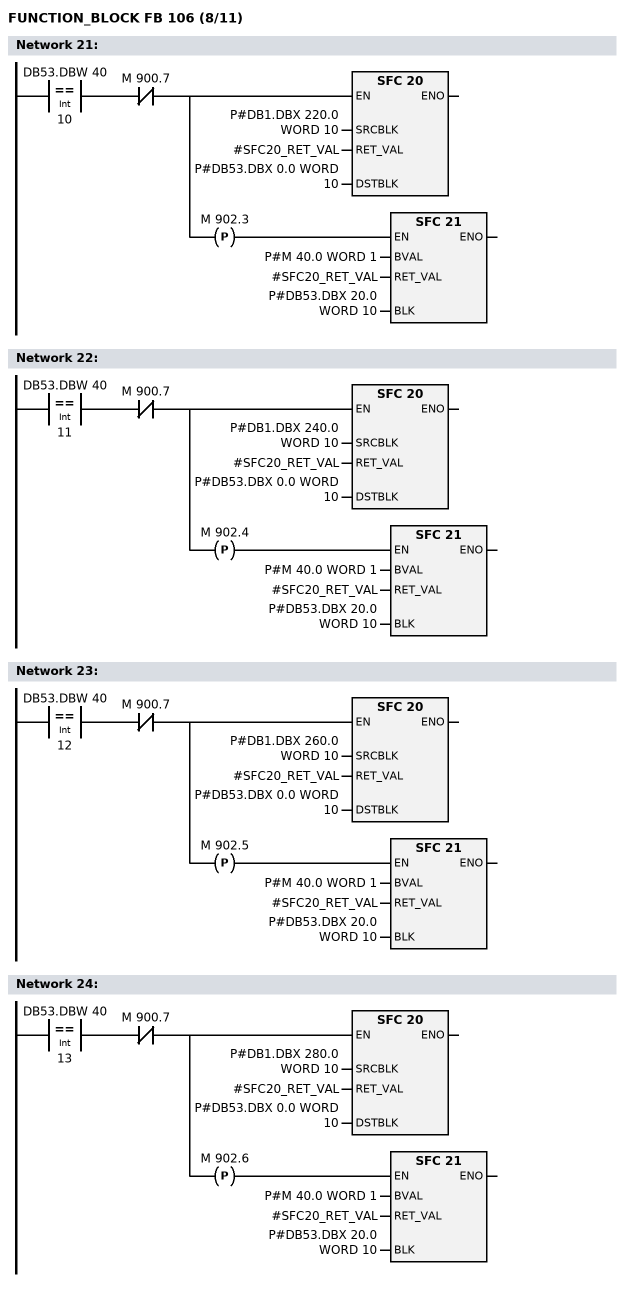

      A(    ;
      L     DB53.DBW   40;
      L     10;
      ==I   ;
      )     ;
      AN    M    900.7;
      =     L      0.0;
      A     L      0.0;
      JNB   _02d;
      CALL SFC   20 (
           SRCBLK                   := P#DB1.DBX 220.0 WORD 10,
           RET_VAL                  := #SFC20_RET_VAL,
           DSTBLK                   := P#DB53.DBX 0.0 WORD 10);
_02d: NOP   0;
      A     L      0.0;
      FP    M    902.3;
      JNB   _02e;
      CALL SFC   21 (
           BVAL                     := P#M 40.0 WORD 1,
           RET_VAL                  := #SFC20_RET_VAL,
           BLK                      := P#DB53.DBX 20.0 WORD 10);
_02e: NOP   0;
NETWORK
TITLE =

      A(    ;
      L     DB53.DBW   40;
      L     11;
      ==I   ;
      )     ;
      AN    M    900.7;
      =     L      0.0;
      A     L      0.0;
      JNB   _02f;
      CALL SFC   20 (
           SRCBLK                   := P#DB1.DBX 240.0 WORD 10,
           RET_VAL                  := #SFC20_RET_VAL,
           DSTBLK                   := P#DB53.DBX 0.0 WORD 10);
_02f: NOP   0;
      A     L      0.0;
      FP    M    902.4;
      JNB   _030;
      CALL SFC   21 (
           BVAL                     := P#M 40.0 WORD 1,
           RET_VAL                  := #SFC20_RET_VAL,
           BLK                      := P#DB53.DBX 20.0 WORD 10);
_030: NOP   0;
NETWORK
TITLE =

      A(    ;
      L     DB53.DBW   40;
      L     12;
      ==I   ;
      )     ;
      AN    M    900.7;
      =     L      0.0;
      A     L      0.0;
      JNB   _031;
      CALL SFC   20 (
           SRCBLK                   := P#DB1.DBX 260.0 WORD 10,
           RET_VAL                  := #SFC20_RET_VAL,
           DSTBLK                   := P#DB53.DBX 0.0 WORD 10);
_031: NOP   0;
      A     L      0.0;
      FP    M    902.5;
      JNB   _032;
      CALL SFC   21 (
           BVAL                     := P#M 40.0 WORD 1,
           RET_VAL                  := #SFC20_RET_VAL,
           BLK                      := P#DB53.DBX 20.0 WORD 10);
_032: NOP   0;
NETWORK
TITLE =

      A(    ;
      L     DB53.DBW   40;
      L     13;
      ==I   ;
      )     ;
      AN    M    900.7;
      =     L      0.0;
      A     L      0.0;
      JNB   _033;
      CALL SFC   20 (
           SRCBLK                   := P#DB1.DBX 280.0 WORD 10,
           RET_VAL                  := #SFC20_RET_VAL,
           DSTBLK                   := P#DB53.DBX 0.0 WORD 10);
_033: NOP   0;
      A     L      0.0;
      FP    M    902.6;
      JNB   _034;
      CALL SFC   21 (
           BVAL                     := P#M 40.0 WORD 1,
           RET_VAL                  := #SFC20_RET_VAL,
           BLK                      := P#DB53.DBX 20.0 WORD 10);
_034: NOP   0;
NETWORK
TITLE =
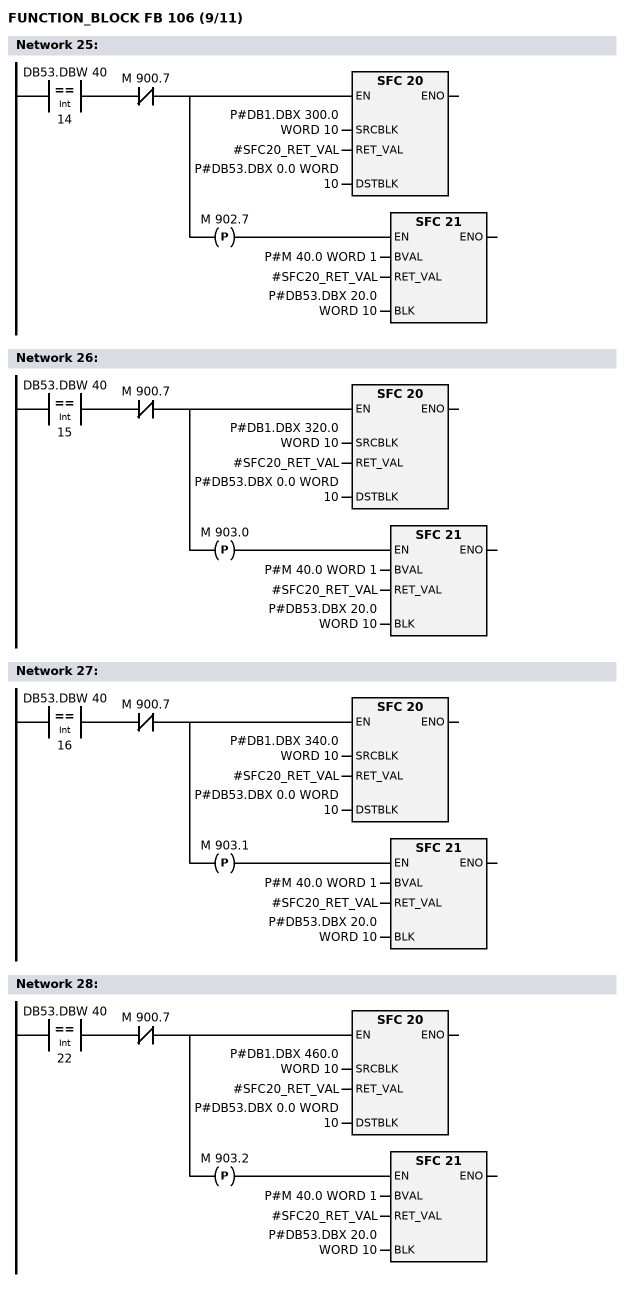

      A(    ;
      L     DB53.DBW   40;
      L     14;
      ==I   ;
      )     ;
      AN    M    900.7;
      =     L      0.0;
      A     L      0.0;
      JNB   _035;
      CALL SFC   20 (
           SRCBLK                   := P#DB1.DBX 300.0 WORD 10,
           RET_VAL                  := #SFC20_RET_VAL,
           DSTBLK                   := P#DB53.DBX 0.0 WORD 10);
_035: NOP   0;
      A     L      0.0;
      FP    M    902.7;
      JNB   _036;
      CALL SFC   21 (
           BVAL                     := P#M 40.0 WORD 1,
           RET_VAL                  := #SFC20_RET_VAL,
           BLK                      := P#DB53.DBX 20.0 WORD 10);
_036: NOP   0;
NETWORK
TITLE =

      A(    ;
      L     DB53.DBW   40;
      L     15;
      ==I   ;
      )     ;
      AN    M    900.7;
      =     L      0.0;
      A     L      0.0;
      JNB   _037;
      CALL SFC   20 (
           SRCBLK                   := P#DB1.DBX 320.0 WORD 10,
           RET_VAL                  := #SFC20_RET_VAL,
           DSTBLK                   := P#DB53.DBX 0.0 WORD 10);
_037: NOP   0;
      A     L      0.0;
      FP    M    903.0;
      JNB   _038;
      CALL SFC   21 (
           BVAL                     := P#M 40.0 WORD 1,
           RET_VAL                  := #SFC20_RET_VAL,
           BLK                      := P#DB53.DBX 20.0 WORD 10);
_038: NOP   0;
NETWORK
TITLE =

      A(    ;
      L     DB53.DBW   40;
      L     16;
      ==I   ;
      )     ;
      AN    M    900.7;
      =     L      0.0;
      A     L      0.0;
      JNB   _039;
      CALL SFC   20 (
           SRCBLK                   := P#DB1.DBX 340.0 WORD 10,
           RET_VAL                  := #SFC20_RET_VAL,
           DSTBLK                   := P#DB53.DBX 0.0 WORD 10);
_039: NOP   0;
      A     L      0.0;
      FP    M    903.1;
      JNB   _03a;
      CALL SFC   21 (
           BVAL                     := P#M 40.0 WORD 1,
           RET_VAL                  := #SFC20_RET_VAL,
           BLK                      := P#DB53.DBX 20.0 WORD 10);
_03a: NOP   0;
NETWORK
TITLE =

      A(    ;
      L     DB53.DBW   40;
      L     22;
      ==I   ;
      )     ;
      AN    M    900.7;
      =     L      0.0;
      A     L      0.0;
      JNB   _03b;
      CALL SFC   20 (
           SRCBLK                   := P#DB1.DBX 460.0 WORD 10,
           RET_VAL                  := #SFC20_RET_VAL,
           DSTBLK                   := P#DB53.DBX 0.0 WORD 10);
_03b: NOP   0;
      A     L      0.0;
      FP    M    903.2;
      JNB   _03c;
      CALL SFC   21 (
           BVAL                     := P#M 40.0 WORD 1,
           RET_VAL                  := #SFC20_RET_VAL,
           BLK                      := P#DB53.DBX 20.0 WORD 10);
_03c: NOP   0;
NETWORK
TITLE =
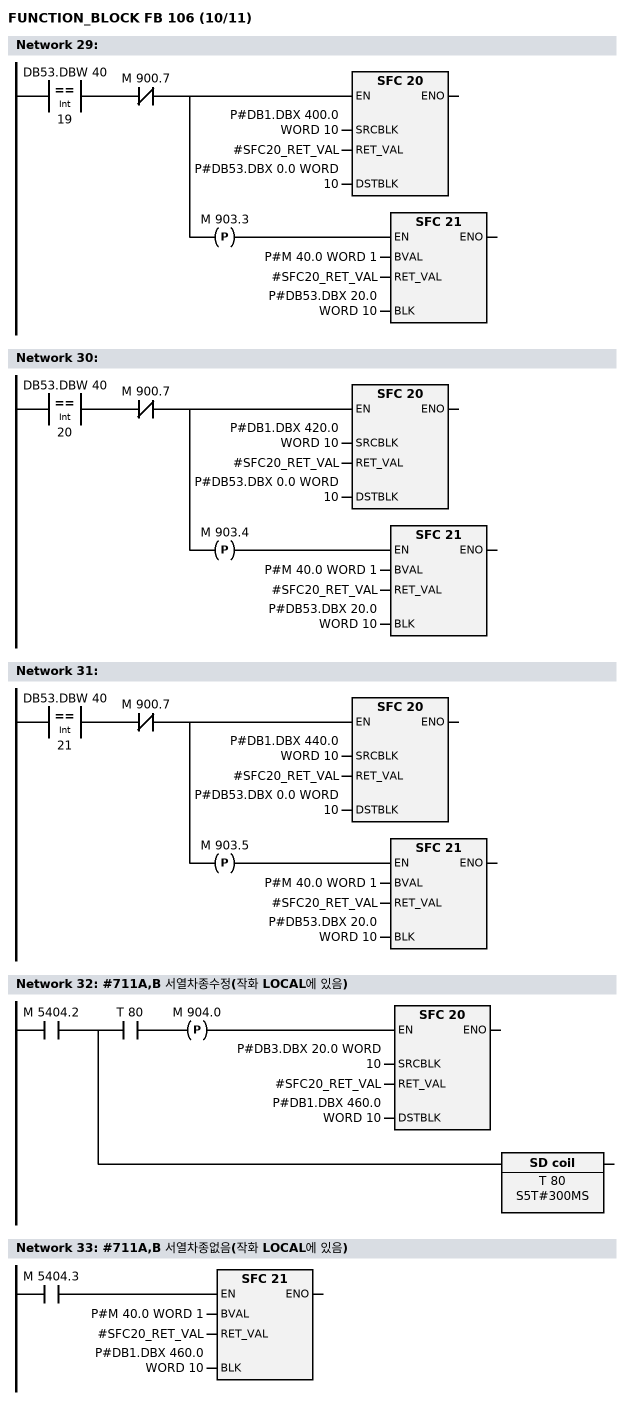

      A(    ;
      L     DB53.DBW   40;
      L     19;
      ==I   ;
      )     ;
      AN    M    900.7;
      =     L      0.0;
      A     L      0.0;
      JNB   _03d;
      CALL SFC   20 (
           SRCBLK                   := P#DB1.DBX 400.0 WORD 10,
           RET_VAL                  := #SFC20_RET_VAL,
           DSTBLK                   := P#DB53.DBX 0.0 WORD 10);
_03d: NOP   0;
      A     L      0.0;
      FP    M    903.3;
      JNB   _03e;
      CALL SFC   21 (
           BVAL                     := P#M 40.0 WORD 1,
           RET_VAL                  := #SFC20_RET_VAL,
           BLK                      := P#DB53.DBX 20.0 WORD 10);
_03e: NOP   0;
NETWORK
TITLE =

      A(    ;
      L     DB53.DBW   40;
      L     20;
      ==I   ;
      )     ;
      AN    M    900.7;
      =     L      0.0;
      A     L      0.0;
      JNB   _03f;
      CALL SFC   20 (
           SRCBLK                   := P#DB1.DBX 420.0 WORD 10,
           RET_VAL                  := #SFC20_RET_VAL,
           DSTBLK                   := P#DB53.DBX 0.0 WORD 10);
_03f: NOP   0;
      A     L      0.0;
      FP    M    903.4;
      JNB   _040;
      CALL SFC   21 (
           BVAL                     := P#M 40.0 WORD 1,
           RET_VAL                  := #SFC20_RET_VAL,
           BLK                      := P#DB53.DBX 20.0 WORD 10);
_040: NOP   0;
NETWORK
TITLE =

      A(    ;
      L     DB53.DBW   40;
      L     21;
      ==I   ;
      )     ;
      AN    M    900.7;
      =     L      0.0;
      A     L      0.0;
      JNB   _041;
      CALL SFC   20 (
           SRCBLK                   := P#DB1.DBX 440.0 WORD 10,
           RET_VAL                  := #SFC20_RET_VAL,
           DSTBLK                   := P#DB53.DBX 0.0 WORD 10);
_041: NOP   0;
      A     L      0.0;
      FP    M    903.5;
      JNB   _042;
      CALL SFC   21 (
           BVAL                     := P#M 40.0 WORD 1,
           RET_VAL                  := #SFC20_RET_VAL,
           BLK                      := P#DB53.DBX 20.0 WORD 10);
_042: NOP   0;
NETWORK
TITLE =#711A,B 서열차종수정(작화 LOCAL에 있음)

      A     M   5404.2;
      =     L      0.0;
      A     L      0.0;
      A     T     80;
      FP    M    904.0;
      JNB   _043;
      CALL SFC   20 (
           SRCBLK                   := P#DB3.DBX 20.0 WORD 10,
           RET_VAL                  := #SFC20_RET_VAL,
           DSTBLK                   := P#DB1.DBX 460.0 WORD 10);
_043: NOP   0;
      A     L      0.0;
      BLD   102;
      L     S5T#300MS;
      SD    T     80;
NETWORK
TITLE =#711A,B 서열차종없음(작화 LOCAL에 있음)

      A     M   5404.3;
      JNB   _044;
      CALL SFC   21 (
           BVAL                     := P#M 40.0 WORD 1,
           RET_VAL                  := #SFC20_RET_VAL,
           BLK                      := P#DB1.DBX 460.0 WORD 10);
_044: NOP   0;
NETWORK
TITLE =#711R1,R2 로보트 차종수정(작화 LOCAL에 있음)
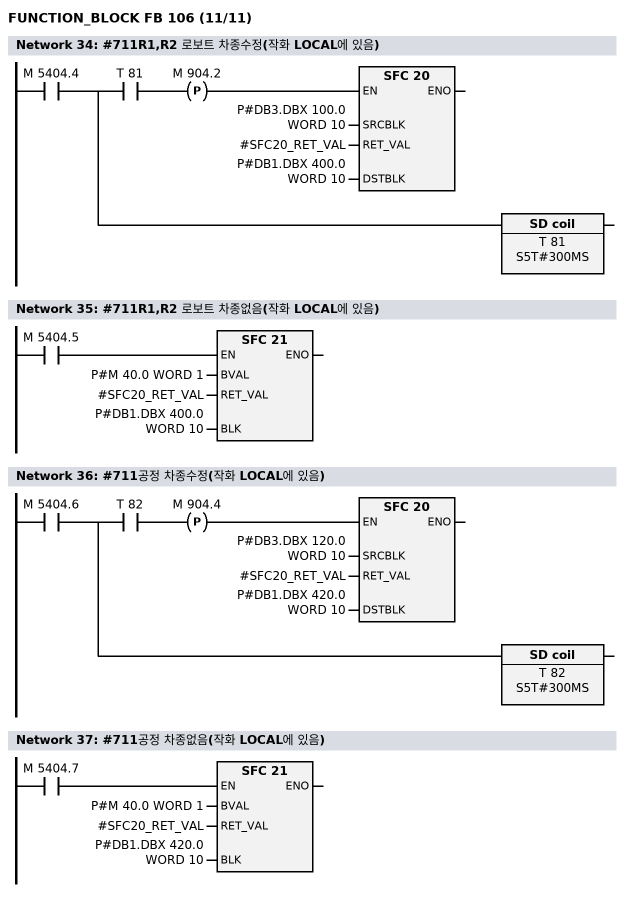

      A     M   5404.4;
      =     L      0.0;
      A     L      0.0;
      A     T     81;
      FP    M    904.2;
      JNB   _045;
      CALL SFC   20 (
           SRCBLK                   := P#DB3.DBX 100.0 WORD 10,
           RET_VAL                  := #SFC20_RET_VAL,
           DSTBLK                   := P#DB1.DBX 400.0 WORD 10);
_045: NOP   0;
      A     L      0.0;
      BLD   102;
      L     S5T#300MS;
      SD    T     81;
NETWORK
TITLE =#711R1,R2 로보트 차종없음(작화 LOCAL에 있음)

      A     M   5404.5;
      JNB   _046;
      CALL SFC   21 (
           BVAL                     := P#M 40.0 WORD 1,
           RET_VAL                  := #SFC20_RET_VAL,
           BLK                      := P#DB1.DBX 400.0 WORD 10);
_046: NOP   0;
NETWORK
TITLE =#711공정 차종수정(작화 LOCAL에 있음)

      A     M   5404.6;
      =     L      0.0;
      A     L      0.0;
      A     T     82;
      FP    M    904.4;
      JNB   _047;
      CALL SFC   20 (
           SRCBLK                   := P#DB3.DBX 120.0 WORD 10,
           RET_VAL                  := #SFC20_RET_VAL,
           DSTBLK                   := P#DB1.DBX 420.0 WORD 10);
_047: NOP   0;
      A     L      0.0;
      BLD   102;
      L     S5T#300MS;
      SD    T     82;
NETWORK
TITLE =#711공정 차종없음(작화 LOCAL에 있음)

      A     M   5404.7;
      JNB   _048;
      CALL SFC   21 (
           BVAL                     := P#M 40.0 WORD 1,
           RET_VAL                  := #SFC20_RET_VAL,
           BLK                      := P#DB1.DBX 420.0 WORD 10);
_048: NOP   0;
END_FUNCTION_BLOCK

DATA_BLOCK DB 106
TITLE =
VERSION : 0.0

 FB 106
BEGIN
   CAR_TYPE_MODIFY.Station := 0;
   CAR_TYPE_MODIFY.HMI_Disp_DB := 0;
   CAR_TYPE_MODIFY.HMI_Disp_Add := 0;
   CAR_TYPE_MODIFY.CType_DB := 0;
   CAR_TYPE_MODIFY.CType_Start_Add := 0;
   CAR_TYPE_MODIFY.Byte_per_Stn := 0;
   CAR_TYPE_MODIFY.M_Modify_OK := FALSE;
   CAR_TYPE_MODIFY.SS_CCR_On := FALSE;
   CAR_TYPE_MODIFY.PB_Set := FALSE;
   CAR_TYPE_MODIFY.PB_Reset := FALSE;
   CAR_TYPE_MODIFY.LP_CCR_On := FALSE;
   CAR_TYPE_MODIFY.LP_Modify_On := FALSE;
   CAR_TYPE_MODIFY.Source_Data := W#16#0;
   CAR_TYPE_MODIFY.Modify_Data := W#16#0;
   CAR_TYPE_MODIFY.Pre_Station := 0;
   CAR_TYPE_MODIFY.Station_PLS := FALSE;
   CAR_TYPE_MODIFY.Source_Add := 0;
   CAR_TYPE_MODIFY.SFC20_Ret := 0;
   CAR_TYPE_MODIFY.Fill_Source := W#16#0;
   SFC20_RET_VAL := 0;
   HMI_CAR_TYPE_V2.Stn_Vin_No := L#0;
   HMI_CAR_TYPE_V2.Stn_Bt_1Word := W#16#0;
   HMI_CAR_TYPE_V2.Stn_Bt_2Word := W#16#0;
   HMI_CAR_TYPE_V2.Stn_Bt_3Word := W#16#0;
   HMI_CAR_TYPE_V2.Stn_Bt_4Word := W#16#0;
   HMI_CAR_TYPE_V2.Stn_Bt_5Word_Sp := W#16#0;
   HMI_CAR_TYPE_V2.Stn_Bt_6Word_Sp := W#16#0;
   HMI_CAR_TYPE_V2.M_BType_On := FALSE;
   HMI_CAR_TYPE_V2.M_BType_None := FALSE;
   HMI_CAR_TYPE_V2.M_Bypass_BType := FALSE;
   HMI_CAR_TYPE_V2.M_BType_TL := FALSE;
   HMI_CAR_TYPE_V2.M_BType_LM := FALSE;
   HMI_CAR_TYPE_V2.M_BType_SP1 := FALSE;
   HMI_CAR_TYPE_V2.M_BType_SP2 := FALSE;
   HMI_CAR_TYPE_V2.M_BType_SP3 := FALSE;
   HMI_CAR_TYPE_V2.M_BType_DOM := FALSE;
   HMI_CAR_TYPE_V2.M_BType_EXP := FALSE;
   HMI_CAR_TYPE_V2.Robot_Prog_No := 0;
   HMI_CAR_TYPE_V2.STN_Btype_1Arr[0] := FALSE;
   HMI_CAR_TYPE_V2.STN_Btype_1Arr[1] := FALSE;
   HMI_CAR_TYPE_V2.STN_Btype_1Arr[2] := FALSE;
   HMI_CAR_TYPE_V2.STN_Btype_1Arr[3] := FALSE;
   HMI_CAR_TYPE_V2.STN_Btype_1Arr[4] := FALSE;
   HMI_CAR_TYPE_V2.STN_Btype_1Arr[5] := FALSE;
   HMI_CAR_TYPE_V2.STN_Btype_1Arr[6] := FALSE;
   HMI_CAR_TYPE_V2.STN_Btype_1Arr[7] := FALSE;
   HMI_CAR_TYPE_V2.STN_Btype_1Arr[8] := FALSE;
   HMI_CAR_TYPE_V2.STN_Btype_1Arr[9] := FALSE;
   HMI_CAR_TYPE_V2.STN_Btype_1Arr[10] := FALSE;
   HMI_CAR_TYPE_V2.STN_Btype_1Arr[11] := FALSE;
   HMI_CAR_TYPE_V2.STN_Btype_1Arr[12] := FALSE;
   HMI_CAR_TYPE_V2.STN_Btype_1Arr[13] := FALSE;
   HMI_CAR_TYPE_V2.STN_Btype_1Arr[14] := FALSE;
   HMI_CAR_TYPE_V2.STN_Btype_1Arr[15] := FALSE;
   HMI_CAR_TYPE_V2.STN_Btype_2Arr[0] := FALSE;
   HMI_CAR_TYPE_V2.STN_Btype_2Arr[1] := FALSE;
   HMI_CAR_TYPE_V2.STN_Btype_2Arr[2] := FALSE;
   HMI_CAR_TYPE_V2.STN_Btype_2Arr[3] := FALSE;
   HMI_CAR_TYPE_V2.STN_Btype_2Arr[4] := FALSE;
   HMI_CAR_TYPE_V2.STN_Btype_2Arr[5] := FALSE;
   HMI_CAR_TYPE_V2.STN_Btype_2Arr[6] := FALSE;
   HMI_CAR_TYPE_V2.STN_Btype_2Arr[7] := FALSE;
   HMI_CAR_TYPE_V2.STN_Btype_2Arr[8] := FALSE;
   HMI_CAR_TYPE_V2.STN_Btype_2Arr[9] := FALSE;
   HMI_CAR_TYPE_V2.STN_Btype_2Arr[10] := FALSE;
   HMI_CAR_TYPE_V2.STN_Btype_2Arr[11] := FALSE;
   HMI_CAR_TYPE_V2.STN_Btype_2Arr[12] := FALSE;
   HMI_CAR_TYPE_V2.STN_Btype_2Arr[13] := FALSE;
   HMI_CAR_TYPE_V2.STN_Btype_2Arr[14] := FALSE;
   HMI_CAR_TYPE_V2.STN_Btype_2Arr[15] := FALSE;
   HMI_CAR_TYPE_V2.STN_Btype_3Arr[0] := FALSE;
   HMI_CAR_TYPE_V2.STN_Btype_3Arr[1] := FALSE;
   HMI_CAR_TYPE_V2.STN_Btype_3Arr[2] := FALSE;
   HMI_CAR_TYPE_V2.STN_Btype_3Arr[3] := FALSE;
   HMI_CAR_TYPE_V2.STN_Btype_3Arr[4] := FALSE;
   HMI_CAR_TYPE_V2.STN_Btype_3Arr[5] := FALSE;
   HMI_CAR_TYPE_V2.STN_Btype_3Arr[6] := FALSE;
   HMI_CAR_TYPE_V2.STN_Btype_3Arr[7] := FALSE;
   HMI_CAR_TYPE_V2.STN_Btype_3Arr[8] := FALSE;
   HMI_CAR_TYPE_V2.STN_Btype_3Arr[9] := FALSE;
   HMI_CAR_TYPE_V2.STN_Btype_3Arr[10] := FALSE;
   HMI_CAR_TYPE_V2.STN_Btype_3Arr[11] := FALSE;
   HMI_CAR_TYPE_V2.STN_Btype_3Arr[12] := FALSE;
   HMI_CAR_TYPE_V2.STN_Btype_3Arr[13] := FALSE;
   HMI_CAR_TYPE_V2.STN_Btype_3Arr[14] := FALSE;
   HMI_CAR_TYPE_V2.STN_Btype_3Arr[15] := FALSE;
   HMI_CAR_TYPE_V2.STN_Btype_4Arr[0] := FALSE;
   HMI_CAR_TYPE_V2.STN_Btype_4Arr[1] := FALSE;
   HMI_CAR_TYPE_V2.STN_Btype_4Arr[2] := FALSE;
   HMI_CAR_TYPE_V2.STN_Btype_4Arr[3] := FALSE;
   HMI_CAR_TYPE_V2.STN_Btype_4Arr[4] := FALSE;
   HMI_CAR_TYPE_V2.STN_Btype_4Arr[5] := FALSE;
   HMI_CAR_TYPE_V2.STN_Btype_4Arr[6] := FALSE;
   HMI_CAR_TYPE_V2.STN_Btype_4Arr[7] := FALSE;
   HMI_CAR_TYPE_V2.STN_Btype_4Arr[8] := FALSE;
   HMI_CAR_TYPE_V2.STN_Btype_4Arr[9] := FALSE;
   HMI_CAR_TYPE_V2.STN_Btype_4Arr[10] := FALSE;
   HMI_CAR_TYPE_V2.STN_Btype_4Arr[11] := FALSE;
   HMI_CAR_TYPE_V2.STN_Btype_4Arr[12] := FALSE;
   HMI_CAR_TYPE_V2.STN_Btype_4Arr[13] := FALSE;
   HMI_CAR_TYPE_V2.STN_Btype_4Arr[14] := FALSE;
   HMI_CAR_TYPE_V2.STN_Btype_4Arr[15] := FALSE;
   HMI_CAR_TYPE_V2.STN_Btype_5Arr[0] := FALSE;
   HMI_CAR_TYPE_V2.STN_Btype_5Arr[1] := FALSE;
   HMI_CAR_TYPE_V2.STN_Btype_5Arr[2] := FALSE;
   HMI_CAR_TYPE_V2.STN_Btype_5Arr[3] := FALSE;
   HMI_CAR_TYPE_V2.STN_Btype_5Arr[4] := FALSE;
   HMI_CAR_TYPE_V2.STN_Btype_5Arr[5] := FALSE;
   HMI_CAR_TYPE_V2.STN_Btype_5Arr[6] := FALSE;
   HMI_CAR_TYPE_V2.STN_Btype_5Arr[7] := FALSE;
   HMI_CAR_TYPE_V2.STN_Btype_5Arr[8] := FALSE;
   HMI_CAR_TYPE_V2.STN_Btype_5Arr[9] := FALSE;
   HMI_CAR_TYPE_V2.STN_Btype_5Arr[10] := FALSE;
   HMI_CAR_TYPE_V2.STN_Btype_5Arr[11] := FALSE;
   HMI_CAR_TYPE_V2.STN_Btype_5Arr[12] := FALSE;
   HMI_CAR_TYPE_V2.STN_Btype_5Arr[13] := FALSE;
   HMI_CAR_TYPE_V2.STN_Btype_5Arr[14] := FALSE;
   HMI_CAR_TYPE_V2.STN_Btype_5Arr[15] := FALSE;
   HMI_CAR_TYPE_V2.STN_Btype_6Arr[0] := FALSE;
   HMI_CAR_TYPE_V2.STN_Btype_6Arr[1] := FALSE;
   HMI_CAR_TYPE_V2.STN_Btype_6Arr[2] := FALSE;
   HMI_CAR_TYPE_V2.STN_Btype_6Arr[3] := FALSE;
   HMI_CAR_TYPE_V2.STN_Btype_6Arr[4] := FALSE;
   HMI_CAR_TYPE_V2.STN_Btype_6Arr[5] := FALSE;
   HMI_CAR_TYPE_V2.STN_Btype_6Arr[6] := FALSE;
   HMI_CAR_TYPE_V2.STN_Btype_6Arr[7] := FALSE;
   HMI_CAR_TYPE_V2.STN_Btype_6Arr[8] := FALSE;
   HMI_CAR_TYPE_V2.STN_Btype_6Arr[9] := FALSE;
   HMI_CAR_TYPE_V2.STN_Btype_6Arr[10] := FALSE;
   HMI_CAR_TYPE_V2.STN_Btype_6Arr[11] := FALSE;
   HMI_CAR_TYPE_V2.STN_Btype_6Arr[12] := FALSE;
   HMI_CAR_TYPE_V2.STN_Btype_6Arr[13] := FALSE;
   HMI_CAR_TYPE_V2.STN_Btype_6Arr[14] := FALSE;
   HMI_CAR_TYPE_V2.STN_Btype_6Arr[15] := FALSE;
   HMI_CAR_TYPE_V2.STN_1st_BT_On := FALSE;
   HMI_CAR_TYPE_V2.STN_2nd_BT_On := FALSE;
   HMI_CAR_TYPE_V2.STN_3rd_BT_On := FALSE;
   HMI_CAR_TYPE_V2.STN_4th_BT_On := FALSE;
   HMI_CAR_TYPE_V2.STN_5th_BT_On := FALSE;
   HMI_CAR_TYPE_V2.STN_6th_BT_On := FALSE;
   HMI_CAR_TYPE_V2.STN_7th_BT_On := FALSE;
   HMI_CAR_TYPE_V2.STN_8th_BT_On := FALSE;
   HMI_CAR_TYPE_V2.STN_9th_BT_On := FALSE;
   HMI_CAR_TYPE_V2.STN_10th_BT_On := FALSE;
   HMI_CAR_TYPE_V2.STN_11th_BT_On := FALSE;
   HMI_CAR_TYPE_V2.STN_12th_BT_On := FALSE;
   HMI_CAR_TYPE_V2.STN_1st_BT_Off := FALSE;
   HMI_CAR_TYPE_V2.BLKMove_Ret := 0;
   HMI_CAR_TYPE_V2.VIN_1BCD := W#16#0;
   HMI_CAR_TYPE_V2.VIN_2BCD := W#16#0;
   HMI_CAR_TYPE_V2.VIN_1Int := 0;
   HMI_CAR_TYPE_V2.VIN_2Int := 0;
END_DATA_BLOCK

FUNCTION FC 106 : VOID
TITLE =
VERSION : 0.1

BEGIN
NETWORK
TITLE =
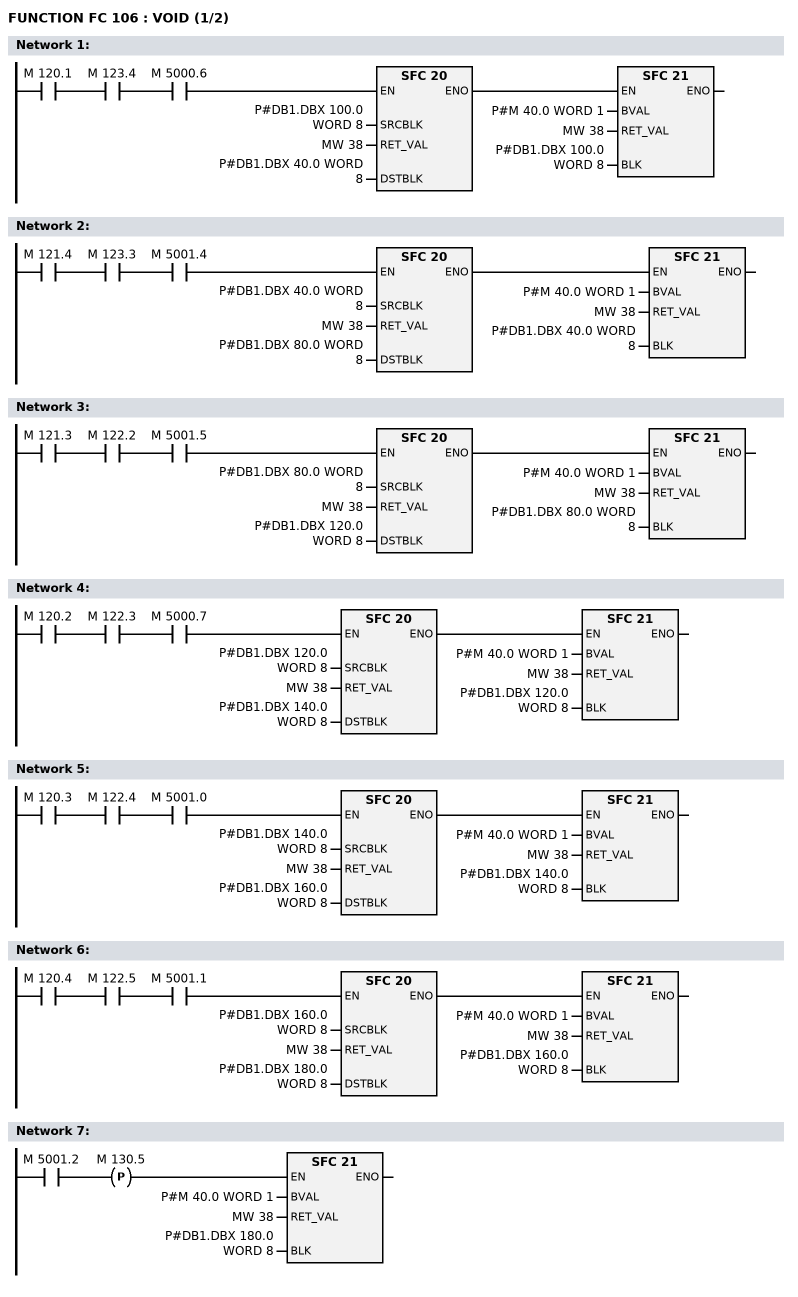

      A(    ;
      A     M    120.1;
      A     M    123.4;
      A     M   5000.6;
      JNB   _001;
      CALL SFC   20 (
           SRCBLK                   := P#DB1.DBX 100.0 WORD 8,
           RET_VAL                  := MW    38,
           DSTBLK                   := P#DB1.DBX 40.0 WORD 8);
_001: A     BR;
      )     ;
      JNB   _002;
      CALL SFC   21 (
           BVAL                     := P#M 40.0 WORD 1,
           RET_VAL                  := MW    38,
           BLK                      := P#DB1.DBX 100.0 WORD 8);
_002: NOP   0;
NETWORK
TITLE =

      A(    ;
      A     M    121.4;
      A     M    123.3;
      A     M   5001.4;
      JNB   _003;
      CALL SFC   20 (
           SRCBLK                   := P#DB1.DBX 40.0 WORD 8,
           RET_VAL                  := MW    38,
           DSTBLK                   := P#DB1.DBX 80.0 WORD 8);
_003: A     BR;
      )     ;
      JNB   _004;
      CALL SFC   21 (
           BVAL                     := P#M 40.0 WORD 1,
           RET_VAL                  := MW    38,
           BLK                      := P#DB1.DBX 40.0 WORD 8);
_004: NOP   0;
NETWORK
TITLE =

      A(    ;
      A     M    121.3;
      A     M    122.2;
      A     M   5001.5;
      JNB   _005;
      CALL SFC   20 (
           SRCBLK                   := P#DB1.DBX 80.0 WORD 8,
           RET_VAL                  := MW    38,
           DSTBLK                   := P#DB1.DBX 120.0 WORD 8);
_005: A     BR;
      )     ;
      JNB   _006;
      CALL SFC   21 (
           BVAL                     := P#M 40.0 WORD 1,
           RET_VAL                  := MW    38,
           BLK                      := P#DB1.DBX 80.0 WORD 8);
_006: NOP   0;
NETWORK
TITLE =

      A(    ;
      A     M    120.2;
      A     M    122.3;
      A     M   5000.7;
      JNB   _007;
      CALL SFC   20 (
           SRCBLK                   := P#DB1.DBX 120.0 WORD 8,
           RET_VAL                  := MW    38,
           DSTBLK                   := P#DB1.DBX 140.0 WORD 8);
_007: A     BR;
      )     ;
      JNB   _008;
      CALL SFC   21 (
           BVAL                     := P#M 40.0 WORD 1,
           RET_VAL                  := MW    38,
           BLK                      := P#DB1.DBX 120.0 WORD 8);
_008: NOP   0;
NETWORK
TITLE =

      A(    ;
      A     M    120.3;
      A     M    122.4;
      A     M   5001.0;
      JNB   _009;
      CALL SFC   20 (
           SRCBLK                   := P#DB1.DBX 140.0 WORD 8,
           RET_VAL                  := MW    38,
           DSTBLK                   := P#DB1.DBX 160.0 WORD 8);
_009: A     BR;
      )     ;
      JNB   _00a;
      CALL SFC   21 (
           BVAL                     := P#M 40.0 WORD 1,
           RET_VAL                  := MW    38,
           BLK                      := P#DB1.DBX 140.0 WORD 8);
_00a: NOP   0;
NETWORK
TITLE =

      A(    ;
      A     M    120.4;
      A     M    122.5;
      A     M   5001.1;
      JNB   _00b;
      CALL SFC   20 (
           SRCBLK                   := P#DB1.DBX 160.0 WORD 8,
           RET_VAL                  := MW    38,
           DSTBLK                   := P#DB1.DBX 180.0 WORD 8);
_00b: A     BR;
      )     ;
      JNB   _00c;
      CALL SFC   21 (
           BVAL                     := P#M 40.0 WORD 1,
           RET_VAL                  := MW    38,
           BLK                      := P#DB1.DBX 160.0 WORD 8);
_00c: NOP   0;
NETWORK
TITLE =

      A     M   5001.2;
      FP    M    130.5;
      JNB   _00d;
      CALL SFC   21 (
           BVAL                     := P#M 40.0 WORD 1,
           RET_VAL                  := MW    38,
           BLK                      := P#DB1.DBX 180.0 WORD 8);
_00d: NOP   0;
NETWORK
TITLE =
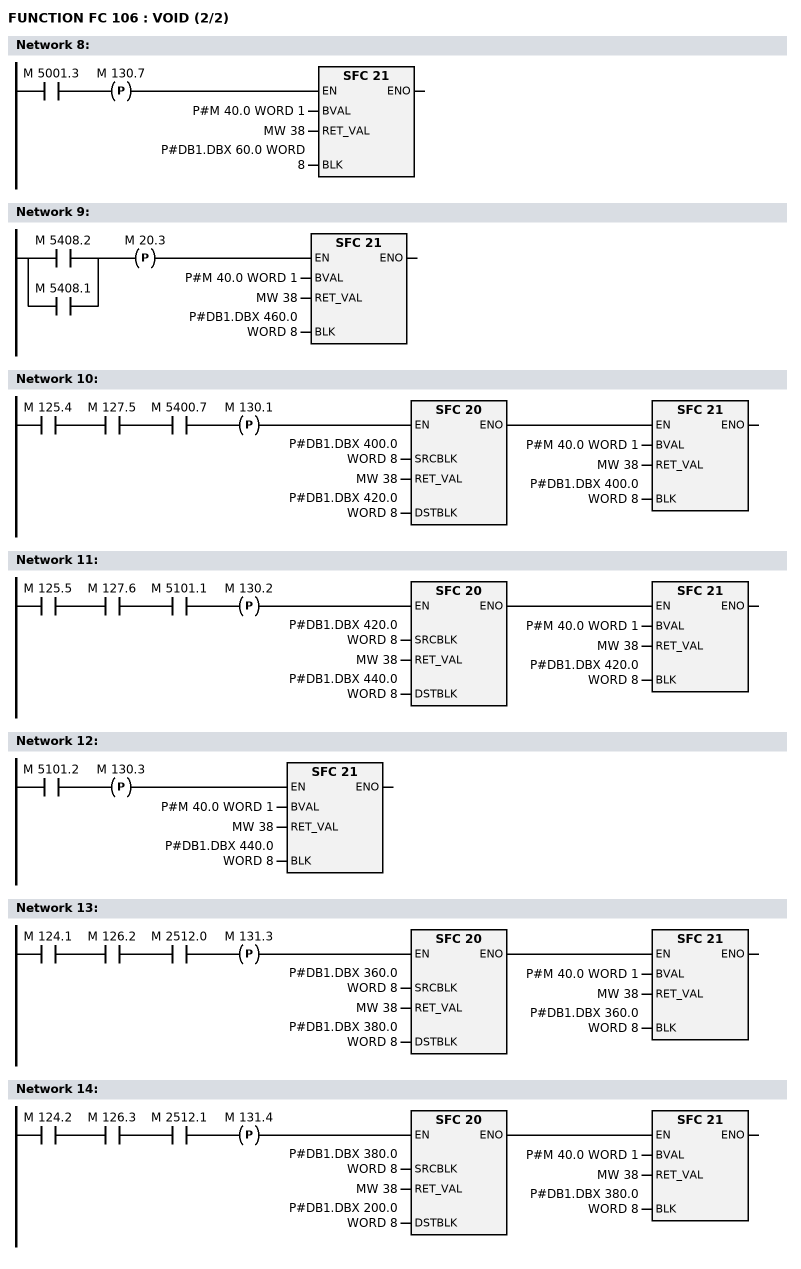

      A     M   5001.3;
      FP    M    130.7;
      JNB   _00e;
      CALL SFC   21 (
           BVAL                     := P#M 40.0 WORD 1,
           RET_VAL                  := MW    38,
           BLK                      := P#DB1.DBX 60.0 WORD 8);
_00e: NOP   0;
NETWORK
TITLE =

      A(    ;
      O     M   5408.2;
      O     M   5408.1;
      )     ;
      FP    M     20.3;
      JNB   _00f;
      CALL SFC   21 (
           BVAL                     := P#M 40.0 WORD 1,
           RET_VAL                  := MW    38,
           BLK                      := P#DB1.DBX 460.0 WORD 8);
_00f: NOP   0;
NETWORK
TITLE =

      A(    ;
      A     M    125.4;
      A     M    127.5;
      A     M   5400.7;
      FP    M    130.1;
      JNB   _010;
      CALL SFC   20 (
           SRCBLK                   := P#DB1.DBX 400.0 WORD 8,
           RET_VAL                  := MW    38,
           DSTBLK                   := P#DB1.DBX 420.0 WORD 8);
_010: A     BR;
      )     ;
      JNB   _011;
      CALL SFC   21 (
           BVAL                     := P#M 40.0 WORD 1,
           RET_VAL                  := MW    38,
           BLK                      := P#DB1.DBX 400.0 WORD 8);
_011: NOP   0;
NETWORK
TITLE =

      A(    ;
      A     M    125.5;
      A     M    127.6;
      A     M   5101.1;
      FP    M    130.2;
      JNB   _012;
      CALL SFC   20 (
           SRCBLK                   := P#DB1.DBX 420.0 WORD 8,
           RET_VAL                  := MW    38,
           DSTBLK                   := P#DB1.DBX 440.0 WORD 8);
_012: A     BR;
      )     ;
      JNB   _013;
      CALL SFC   21 (
           BVAL                     := P#M 40.0 WORD 1,
           RET_VAL                  := MW    38,
           BLK                      := P#DB1.DBX 420.0 WORD 8);
_013: NOP   0;
NETWORK
TITLE =

      A     M   5101.2;
      FP    M    130.3;
      JNB   _014;
      CALL SFC   21 (
           BVAL                     := P#M 40.0 WORD 1,
           RET_VAL                  := MW    38,
           BLK                      := P#DB1.DBX 440.0 WORD 8);
_014: NOP   0;
NETWORK
TITLE =

      A(    ;
      A     M    124.1;
      A     M    126.2;
      A     M   2512.0;
      FP    M    131.3;
      JNB   _015;
      CALL SFC   20 (
           SRCBLK                   := P#DB1.DBX 360.0 WORD 8,
           RET_VAL                  := MW    38,
           DSTBLK                   := P#DB1.DBX 380.0 WORD 8);
_015: A     BR;
      )     ;
      JNB   _016;
      CALL SFC   21 (
           BVAL                     := P#M 40.0 WORD 1,
           RET_VAL                  := MW    38,
           BLK                      := P#DB1.DBX 360.0 WORD 8);
_016: NOP   0;
NETWORK
TITLE =

      A(    ;
      A     M    124.2;
      A     M    126.3;
      A     M   2512.1;
      FP    M    131.4;
      JNB   _017;
      CALL SFC   20 (
           SRCBLK                   := P#DB1.DBX 380.0 WORD 8,
           RET_VAL                  := MW    38,
           DSTBLK                   := P#DB1.DBX 200.0 WORD 8);
_017: A     BR;
      )     ;
      JNB   _018;
      CALL SFC   21 (
           BVAL                     := P#M 40.0 WORD 1,
           RET_VAL                  := MW    38,
           BLK                      := P#DB1.DBX 380.0 WORD 8);
_018: NOP   0;
NETWORK
TITLE =

      A     M    508.6;
      FP    M    131.5;
      =     L      0.0;
      A(    ;
      A     L      0.0;
      JNB   _019;
      CALL SFC   20 (
           SRCBLK                   := P#DB1.DBX 300.0 WORD 8,
           RET_VAL                  := MW    38,
           DSTBLK                   := P#DB1.DBX 320.0 WORD 8);
_019: A     BR;
      )     ;
      JNB   _01a;
      CALL SFC   20 (
           SRCBLK                   := P#DB1.DBX 280.0 WORD 8,
           RET_VAL                  := MW    38,
           DSTBLK                   := P#DB1.DBX 300.0 WORD 8);
_01a: NOP   0;
      A(    ;
      A     L      0.0;
      JNB   _01b;
      CALL SFC   20 (
           SRCBLK                   := P#DB1.DBX 260.0 WORD 8,
           RET_VAL                  := MW    38,
           DSTBLK                   := P#DB1.DBX 280.0 WORD 8);
_01b: A     BR;
      )     ;
      JNB   _01c;
      CALL SFC   20 (
           SRCBLK                   := P#DB1.DBX 240.0 WORD 8,
           RET_VAL                  := MW    38,
           DSTBLK                   := P#DB1.DBX 260.0 WORD 8);
_01c: NOP   0;
      A(    ;
      A     L      0.0;
      JNB   _01d;
      CALL SFC   20 (
           SRCBLK                   := P#DB1.DBX 220.0 WORD 8,
           RET_VAL                  := MW    38,
           DSTBLK                   := P#DB1.DBX 240.0 WORD 8);
_01d: A     BR;
      )     ;
      JNB   _01e;
      CALL SFC   20 (
           SRCBLK                   := P#DB1.DBX 200.0 WORD 8,
           RET_VAL                  := MW    38,
           DSTBLK                   := P#DB1.DBX 220.0 WORD 8);
_01e: NOP   0;
      A     L      0.0;
      JNB   _01f;
      CALL SFC   21 (
           BVAL                     := P#M 40.0 WORD 1,
           RET_VAL                  := MW    38,
           BLK                      := P#DB1.DBX 200.0 WORD 8);
_01f: NOP   0;
NETWORK
TITLE =
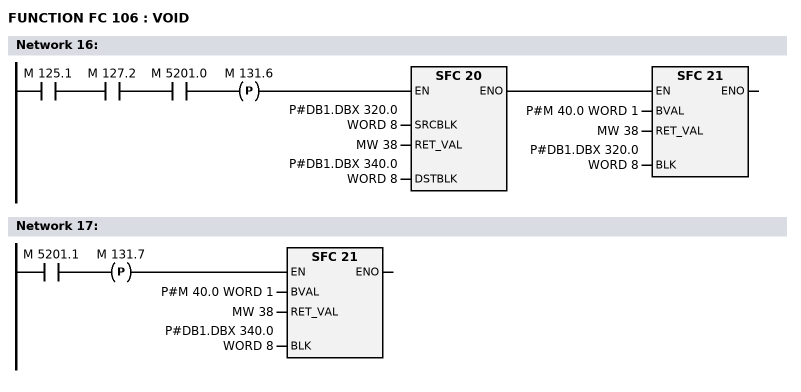

      A(    ;
      A     M    125.1;
      A     M    127.2;
      A     M   5201.0;
      FP    M    131.6;
      JNB   _020;
      CALL SFC   20 (
           SRCBLK                   := P#DB1.DBX 320.0 WORD 8,
           RET_VAL                  := MW    38,
           DSTBLK                   := P#DB1.DBX 340.0 WORD 8);
_020: A     BR;
      )     ;
      JNB   _021;
      CALL SFC   21 (
           BVAL                     := P#M 40.0 WORD 1,
           RET_VAL                  := MW    38,
           BLK                      := P#DB1.DBX 320.0 WORD 8);
_021: NOP   0;
NETWORK
TITLE =

      A     M   5201.1;
      FP    M    131.7;
      JNB   _022;
      CALL SFC   21 (
           BVAL                     := P#M 40.0 WORD 1,
           RET_VAL                  := MW    38,
           BLK                      := P#DB1.DBX 340.0 WORD 8);
_022: NOP   0;
END_FUNCTION

FUNCTION_BLOCK FB 107
TITLE =
VERSION : 0.1


VAR
  O_TRV_CT : FB 500;
  S702_CT : FB 500;
  S703_CT : FB 500;
  S704_CT : FB 500;
  S705_CT : FB 500;
  S706_CT : FB 500;
  S707_CT : FB 500;
  S708_CT : FB 500;
  UP_DL_CT : FB 500;
  ITRV_CT : FB 500;
  ALL_LINE_CT : FB 500;
END_VAR
BEGIN
NETWORK
TITLE =
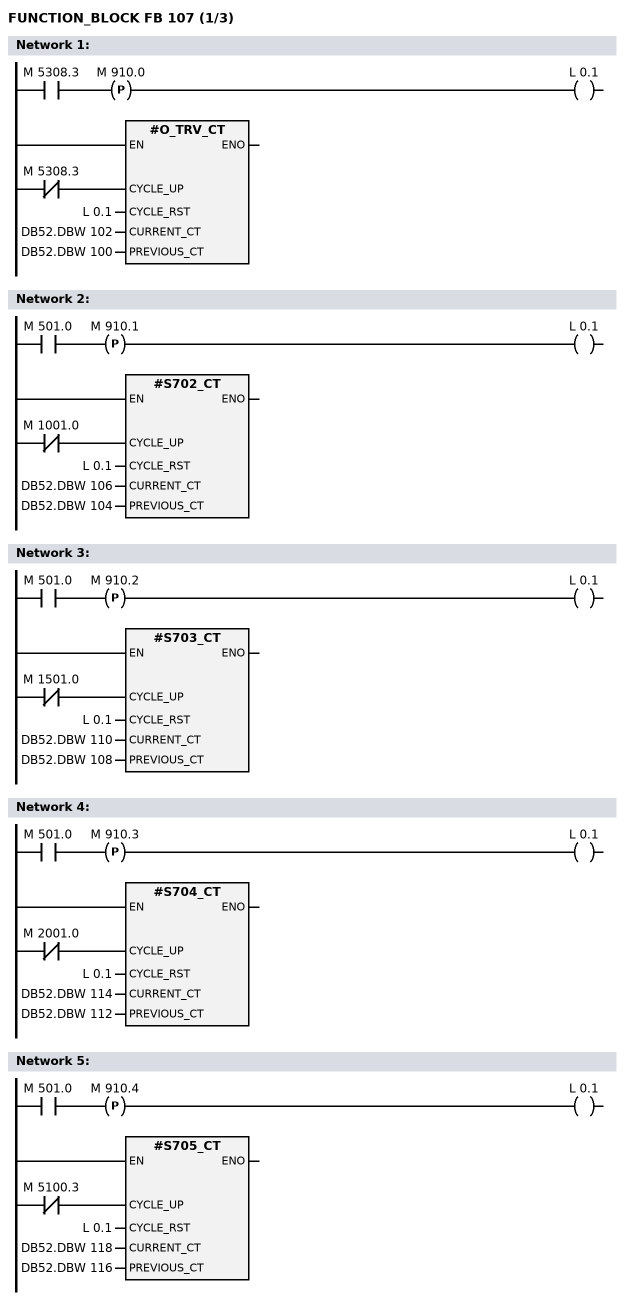

      AN    M   5308.3;
      =     L      0.0;
      BLD   103;
      A     M   5308.3;
      FP    M    910.0;
      =     L      0.1;
      BLD   103;
      CALL #O_TRV_CT (
           CYCLE_UP                 := L      0.0,
           CYCLE_RST                := L      0.1,
           CURRENT_CT               := DB52.DBW  102,
           PREVIOUS_CT              := DB52.DBW  100);
      NOP   0;
NETWORK
TITLE =

      AN    M   1001.0;
      =     L      0.0;
      BLD   103;
      A     M    501.0;
      FP    M    910.1;
      =     L      0.1;
      BLD   103;
      CALL #S702_CT (
           CYCLE_UP                 := L      0.0,
           CYCLE_RST                := L      0.1,
           CURRENT_CT               := DB52.DBW  106,
           PREVIOUS_CT              := DB52.DBW  104);
      NOP   0;
NETWORK
TITLE =

      AN    M   1501.0;
      =     L      0.0;
      BLD   103;
      A     M    501.0;
      FP    M    910.2;
      =     L      0.1;
      BLD   103;
      CALL #S703_CT (
           CYCLE_UP                 := L      0.0,
           CYCLE_RST                := L      0.1,
           CURRENT_CT               := DB52.DBW  110,
           PREVIOUS_CT              := DB52.DBW  108);
      NOP   0;
NETWORK
TITLE =

      AN    M   2001.0;
      =     L      0.0;
      BLD   103;
      A     M    501.0;
      FP    M    910.3;
      =     L      0.1;
      BLD   103;
      CALL #S704_CT (
           CYCLE_UP                 := L      0.0,
           CYCLE_RST                := L      0.1,
           CURRENT_CT               := DB52.DBW  114,
           PREVIOUS_CT              := DB52.DBW  112);
      NOP   0;
NETWORK
TITLE =

      AN    M   5100.3;
      =     L      0.0;
      BLD   103;
      A     M    501.0;
      FP    M    910.4;
      =     L      0.1;
      BLD   103;
      CALL #S705_CT (
           CYCLE_UP                 := L      0.0,
           CYCLE_RST                := L      0.1,
           CURRENT_CT               := DB52.DBW  118,
           PREVIOUS_CT              := DB52.DBW  116);
      NOP   0;
NETWORK
TITLE =
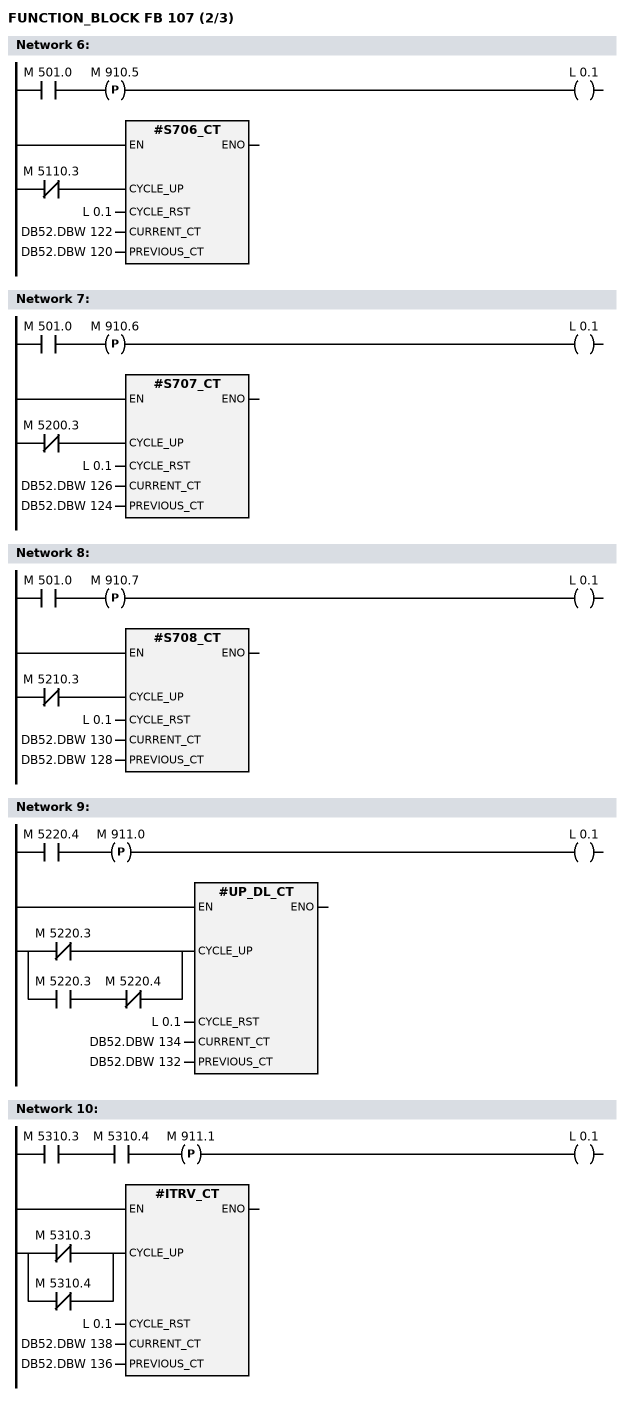

      AN    M   5110.3;
      =     L      0.0;
      BLD   103;
      A     M    501.0;
      FP    M    910.5;
      =     L      0.1;
      BLD   103;
      CALL #S706_CT (
           CYCLE_UP                 := L      0.0,
           CYCLE_RST                := L      0.1,
           CURRENT_CT               := DB52.DBW  122,
           PREVIOUS_CT              := DB52.DBW  120);
      NOP   0;
NETWORK
TITLE =

      AN    M   5200.3;
      =     L      0.0;
      BLD   103;
      A     M    501.0;
      FP    M    910.6;
      =     L      0.1;
      BLD   103;
      CALL #S707_CT (
           CYCLE_UP                 := L      0.0,
           CYCLE_RST                := L      0.1,
           CURRENT_CT               := DB52.DBW  126,
           PREVIOUS_CT              := DB52.DBW  124);
      NOP   0;
NETWORK
TITLE =

      AN    M   5210.3;
      =     L      0.0;
      BLD   103;
      A     M    501.0;
      FP    M    910.7;
      =     L      0.1;
      BLD   103;
      CALL #S708_CT (
           CYCLE_UP                 := L      0.0,
           CYCLE_RST                := L      0.1,
           CURRENT_CT               := DB52.DBW  130,
           PREVIOUS_CT              := DB52.DBW  128);
      NOP   0;
NETWORK
TITLE =

      A(    ;
      ON    M   5220.3;
      O     ;
      A     M   5220.3;
      AN    M   5220.4;
      )     ;
      =     L      0.0;
      BLD   103;
      A     M   5220.4;
      FP    M    911.0;
      =     L      0.1;
      BLD   103;
      CALL #UP_DL_CT (
           CYCLE_UP                 := L      0.0,
           CYCLE_RST                := L      0.1,
           CURRENT_CT               := DB52.DBW  134,
           PREVIOUS_CT              := DB52.DBW  132);
      NOP   0;
NETWORK
TITLE =

      A(    ;
      ON    M   5310.3;
      ON    M   5310.4;
      )     ;
      =     L      0.0;
      BLD   103;
      A     M   5310.3;
      A     M   5310.4;
      FP    M    911.1;
      =     L      0.1;
      BLD   103;
      CALL #ITRV_CT (
           CYCLE_UP                 := L      0.0,
           CYCLE_RST                := L      0.1,
           CURRENT_CT               := DB52.DBW  138,
           PREVIOUS_CT              := DB52.DBW  136);
      NOP   0;
NETWORK
TITLE =
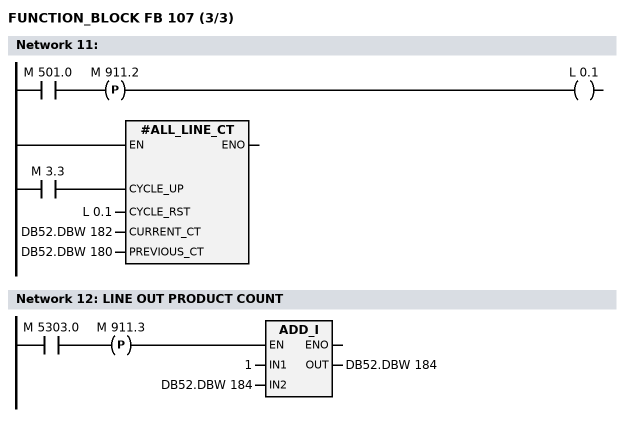

      A     M      3.3;
      =     L      0.0;
      BLD   103;
      A     M    501.0;
      FP    M    911.2;
      =     L      0.1;
      BLD   103;
      CALL #ALL_LINE_CT (
           CYCLE_UP                 := L      0.0,
           CYCLE_RST                := L      0.1,
           CURRENT_CT               := DB52.DBW  182,
           PREVIOUS_CT              := DB52.DBW  180);
      NOP   0;
NETWORK
TITLE =LINE OUT PRODUCT COUNT

      A     M   5303.0;
      FP    M    911.3;
      JNB   _001;
      L     1;
      L     DB52.DBW  184;
      +I    ;
      T     DB52.DBW  184;
_001: NOP   0;
END_FUNCTION_BLOCK

DATA_BLOCK DB 107
TITLE =
VERSION : 0.0

 FB 107
BEGIN
   O_TRV_CT.CYCLE_UP := FALSE;
   O_TRV_CT.CYCLE_RST := FALSE;
   O_TRV_CT.CURRENT_CT := 0;
   O_TRV_CT.PREVIOUS_CT := 0;
   O_TRV_CT.CURRENT := 0;
   O_TRV_CT.PREVIOUS := 0;
   O_TRV_CT.CYCLE_UP_PLS := FALSE;
   O_TRV_CT.CYCLE_RST_PLS := FALSE;
   O_TRV_CT.CYCLE_OVER_PLS := FALSE;
   S702_CT.CYCLE_UP := FALSE;
   S702_CT.CYCLE_RST := FALSE;
   S702_CT.CURRENT_CT := 0;
   S702_CT.PREVIOUS_CT := 0;
   S702_CT.CURRENT := 0;
   S702_CT.PREVIOUS := 0;
   S702_CT.CYCLE_UP_PLS := FALSE;
   S702_CT.CYCLE_RST_PLS := FALSE;
   S702_CT.CYCLE_OVER_PLS := FALSE;
   S703_CT.CYCLE_UP := FALSE;
   S703_CT.CYCLE_RST := FALSE;
   S703_CT.CURRENT_CT := 0;
   S703_CT.PREVIOUS_CT := 0;
   S703_CT.CURRENT := 0;
   S703_CT.PREVIOUS := 0;
   S703_CT.CYCLE_UP_PLS := FALSE;
   S703_CT.CYCLE_RST_PLS := FALSE;
   S703_CT.CYCLE_OVER_PLS := FALSE;
   S704_CT.CYCLE_UP := FALSE;
   S704_CT.CYCLE_RST := FALSE;
   S704_CT.CURRENT_CT := 0;
   S704_CT.PREVIOUS_CT := 0;
   S704_CT.CURRENT := 0;
   S704_CT.PREVIOUS := 0;
   S704_CT.CYCLE_UP_PLS := FALSE;
   S704_CT.CYCLE_RST_PLS := FALSE;
   S704_CT.CYCLE_OVER_PLS := FALSE;
   S705_CT.CYCLE_UP := FALSE;
   S705_CT.CYCLE_RST := FALSE;
   S705_CT.CURRENT_CT := 0;
   S705_CT.PREVIOUS_CT := 0;
   S705_CT.CURRENT := 0;
   S705_CT.PREVIOUS := 0;
   S705_CT.CYCLE_UP_PLS := FALSE;
   S705_CT.CYCLE_RST_PLS := FALSE;
   S705_CT.CYCLE_OVER_PLS := FALSE;
   S706_CT.CYCLE_UP := FALSE;
   S706_CT.CYCLE_RST := FALSE;
   S706_CT.CURRENT_CT := 0;
   S706_CT.PREVIOUS_CT := 0;
   S706_CT.CURRENT := 0;
   S706_CT.PREVIOUS := 0;
   S706_CT.CYCLE_UP_PLS := FALSE;
   S706_CT.CYCLE_RST_PLS := FALSE;
   S706_CT.CYCLE_OVER_PLS := FALSE;
   S707_CT.CYCLE_UP := FALSE;
   S707_CT.CYCLE_RST := FALSE;
   S707_CT.CURRENT_CT := 0;
   S707_CT.PREVIOUS_CT := 0;
   S707_CT.CURRENT := 0;
   S707_CT.PREVIOUS := 0;
   S707_CT.CYCLE_UP_PLS := FALSE;
   S707_CT.CYCLE_RST_PLS := FALSE;
   S707_CT.CYCLE_OVER_PLS := FALSE;
   S708_CT.CYCLE_UP := FALSE;
   S708_CT.CYCLE_RST := FALSE;
   S708_CT.CURRENT_CT := 0;
   S708_CT.PREVIOUS_CT := 0;
   S708_CT.CURRENT := 0;
   S708_CT.PREVIOUS := 0;
   S708_CT.CYCLE_UP_PLS := FALSE;
   S708_CT.CYCLE_RST_PLS := FALSE;
   S708_CT.CYCLE_OVER_PLS := FALSE;
   UP_DL_CT.CYCLE_UP := FALSE;
   UP_DL_CT.CYCLE_RST := FALSE;
   UP_DL_CT.CURRENT_CT := 0;
   UP_DL_CT.PREVIOUS_CT := 0;
   UP_DL_CT.CURRENT := 0;
   UP_DL_CT.PREVIOUS := 0;
   UP_DL_CT.CYCLE_UP_PLS := FALSE;
   UP_DL_CT.CYCLE_RST_PLS := FALSE;
   UP_DL_CT.CYCLE_OVER_PLS := FALSE;
   ITRV_CT.CYCLE_UP := FALSE;
   ITRV_CT.CYCLE_RST := FALSE;
   ITRV_CT.CURRENT_CT := 0;
   ITRV_CT.PREVIOUS_CT := 0;
   ITRV_CT.CURRENT := 0;
   ITRV_CT.PREVIOUS := 0;
   ITRV_CT.CYCLE_UP_PLS := FALSE;
   ITRV_CT.CYCLE_RST_PLS := FALSE;
   ITRV_CT.CYCLE_OVER_PLS := FALSE;
   ALL_LINE_CT.CYCLE_UP := FALSE;
   ALL_LINE_CT.CYCLE_RST := FALSE;
   ALL_LINE_CT.CURRENT_CT := 0;
   ALL_LINE_CT.PREVIOUS_CT := 0;
   ALL_LINE_CT.CURRENT := 0;
   ALL_LINE_CT.PREVIOUS := 0;
   ALL_LINE_CT.CYCLE_UP_PLS := FALSE;
   ALL_LINE_CT.CYCLE_RST_PLS := FALSE;
   ALL_LINE_CT.CYCLE_OVER_PLS := FALSE;
END_DATA_BLOCK

FUNCTION FC 107 : VOID
TITLE =
VERSION : 0.1

BEGIN
NETWORK
TITLE =
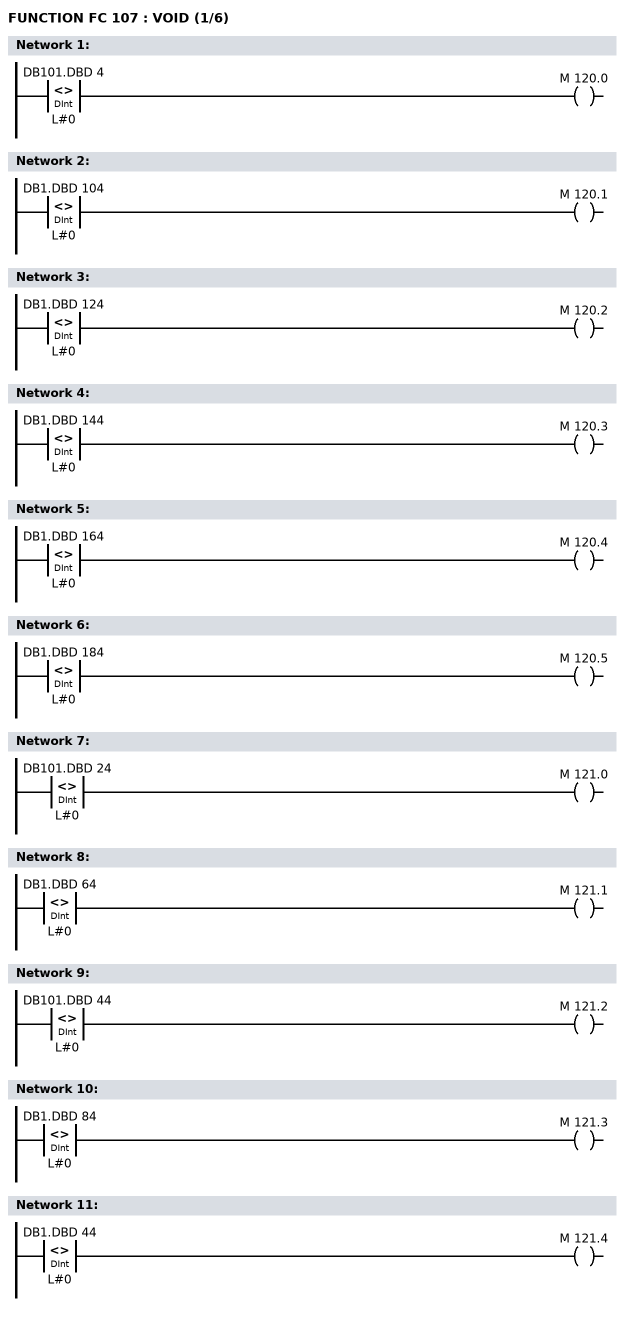

      L     DB101.DBD    4;
      L     L#0;
      <>D   ;
      =     M    120.0;
NETWORK
TITLE =

      L     DB1.DBD  104;
      L     L#0;
      <>D   ;
      =     M    120.1;
NETWORK
TITLE =

      L     DB1.DBD  124;
      L     L#0;
      <>D   ;
      =     M    120.2;
NETWORK
TITLE =

      L     DB1.DBD  144;
      L     L#0;
      <>D   ;
      =     M    120.3;
NETWORK
TITLE =

      L     DB1.DBD  164;
      L     L#0;
      <>D   ;
      =     M    120.4;
NETWORK
TITLE =

      L     DB1.DBD  184;
      L     L#0;
      <>D   ;
      =     M    120.5;
NETWORK
TITLE =

      L     DB101.DBD   24;
      L     L#0;
      <>D   ;
      =     M    121.0;
NETWORK
TITLE =

      L     DB1.DBD   64;
      L     L#0;
      <>D   ;
      =     M    121.1;
NETWORK
TITLE =

      L     DB101.DBD   44;
      L     L#0;
      <>D   ;
      =     M    121.2;
NETWORK
TITLE =

      L     DB1.DBD   84;
      L     L#0;
      <>D   ;
      =     M    121.3;
NETWORK
TITLE =

      L     DB1.DBD   44;
      L     L#0;
      <>D   ;
      =     M    121.4;
NETWORK
TITLE =
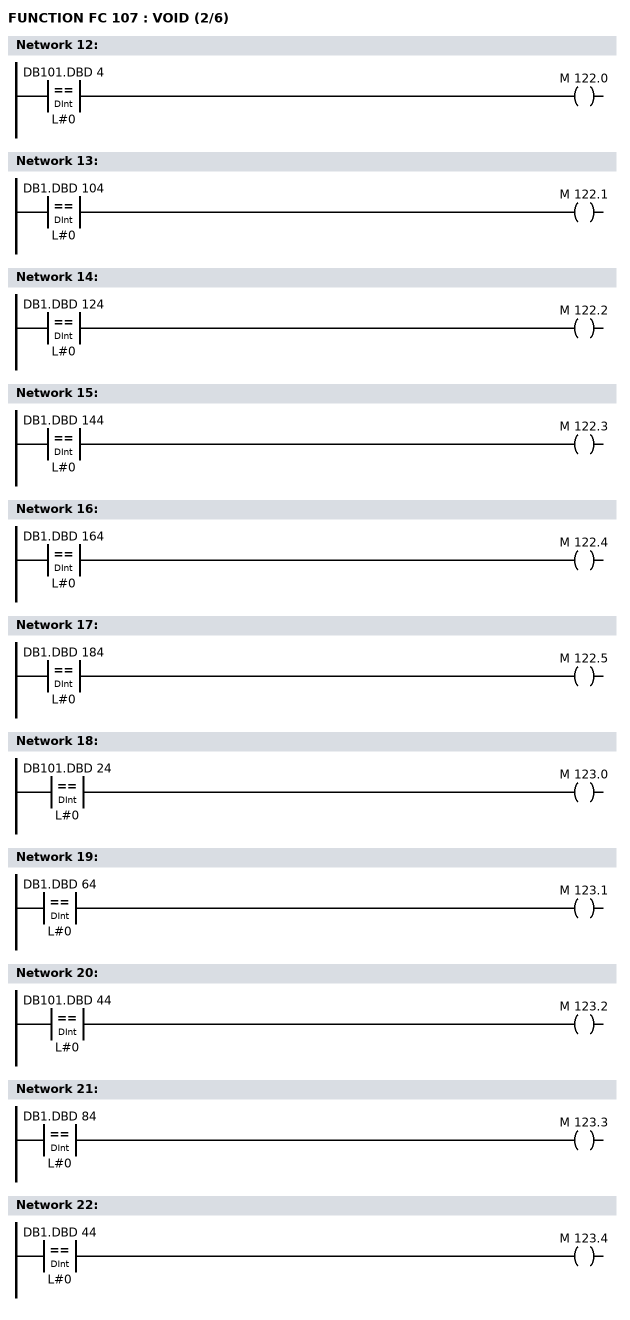

      L     DB101.DBD    4;
      L     L#0;
      ==D   ;
      =     M    122.0;
NETWORK
TITLE =

      L     DB1.DBD  104;
      L     L#0;
      ==D   ;
      =     M    122.1;
NETWORK
TITLE =

      L     DB1.DBD  124;
      L     L#0;
      ==D   ;
      =     M    122.2;
NETWORK
TITLE =

      L     DB1.DBD  144;
      L     L#0;
      ==D   ;
      =     M    122.3;
NETWORK
TITLE =

      L     DB1.DBD  164;
      L     L#0;
      ==D   ;
      =     M    122.4;
NETWORK
TITLE =

      L     DB1.DBD  184;
      L     L#0;
      ==D   ;
      =     M    122.5;
NETWORK
TITLE =

      L     DB101.DBD   24;
      L     L#0;
      ==D   ;
      =     M    123.0;
NETWORK
TITLE =

      L     DB1.DBD   64;
      L     L#0;
      ==D   ;
      =     M    123.1;
NETWORK
TITLE =

      L     DB101.DBD   44;
      L     L#0;
      ==D   ;
      =     M    123.2;
NETWORK
TITLE =

      L     DB1.DBD   84;
      L     L#0;
      ==D   ;
      =     M    123.3;
NETWORK
TITLE =

      L     DB1.DBD   44;
      L     L#0;
      ==D   ;
      =     M    123.4;
NETWORK
TITLE =
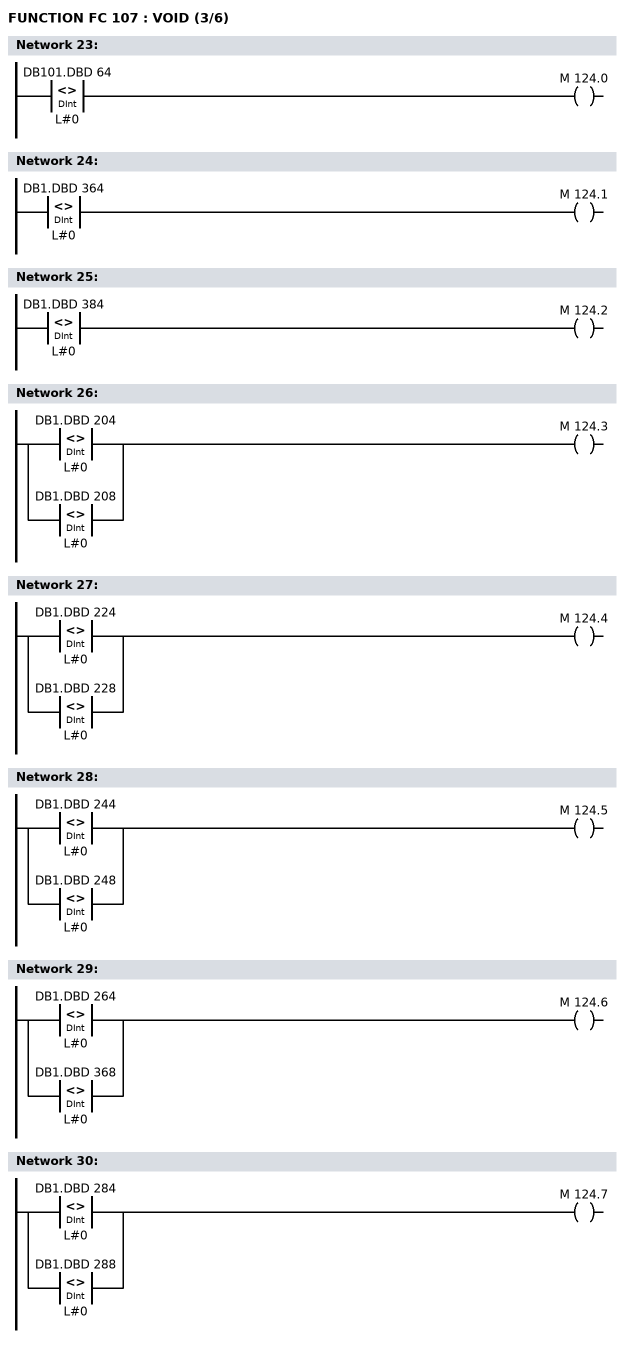

      L     DB101.DBD   64;
      L     L#0;
      <>D   ;
      =     M    124.0;
NETWORK
TITLE =

      L     DB1.DBD  364;
      L     L#0;
      <>D   ;
      =     M    124.1;
NETWORK
TITLE =

      L     DB1.DBD  384;
      L     L#0;
      <>D   ;
      =     M    124.2;
NETWORK
TITLE =

      O(    ;
      L     DB1.DBD  204;
      L     L#0;
      <>D   ;
      )     ;
      O(    ;
      L     DB1.DBD  208;
      L     L#0;
      <>D   ;
      )     ;
      =     M    124.3;
NETWORK
TITLE =

      O(    ;
      L     DB1.DBD  224;
      L     L#0;
      <>D   ;
      )     ;
      O(    ;
      L     DB1.DBD  228;
      L     L#0;
      <>D   ;
      )     ;
      =     M    124.4;
NETWORK
TITLE =

      O(    ;
      L     DB1.DBD  244;
      L     L#0;
      <>D   ;
      )     ;
      O(    ;
      L     DB1.DBD  248;
      L     L#0;
      <>D   ;
      )     ;
      =     M    124.5;
NETWORK
TITLE =

      O(    ;
      L     DB1.DBD  264;
      L     L#0;
      <>D   ;
      )     ;
      O(    ;
      L     DB1.DBD  368;
      L     L#0;
      <>D   ;
      )     ;
      =     M    124.6;
NETWORK
TITLE =

      O(    ;
      L     DB1.DBD  284;
      L     L#0;
      <>D   ;
      )     ;
      O(    ;
      L     DB1.DBD  288;
      L     L#0;
      <>D   ;
      )     ;
      =     M    124.7;
NETWORK
TITLE =
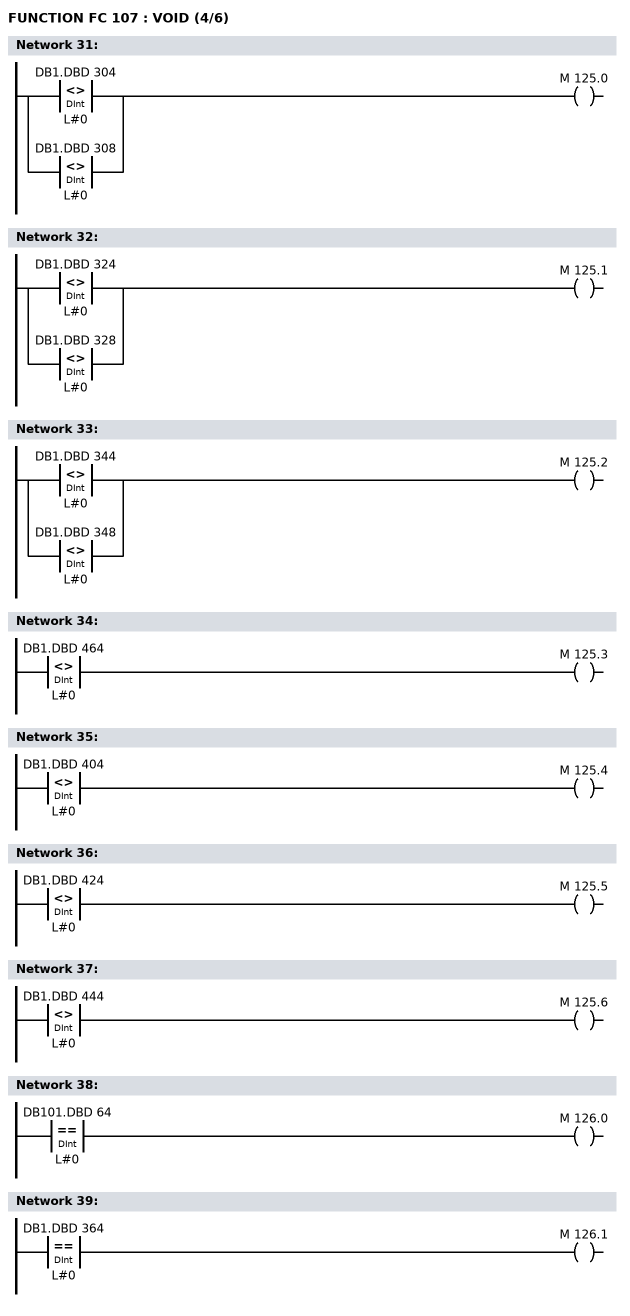

      O(    ;
      L     DB1.DBD  304;
      L     L#0;
      <>D   ;
      )     ;
      O(    ;
      L     DB1.DBD  308;
      L     L#0;
      <>D   ;
      )     ;
      =     M    125.0;
NETWORK
TITLE =

      O(    ;
      L     DB1.DBD  324;
      L     L#0;
      <>D   ;
      )     ;
      O(    ;
      L     DB1.DBD  328;
      L     L#0;
      <>D   ;
      )     ;
      =     M    125.1;
NETWORK
TITLE =

      O(    ;
      L     DB1.DBD  344;
      L     L#0;
      <>D   ;
      )     ;
      O(    ;
      L     DB1.DBD  348;
      L     L#0;
      <>D   ;
      )     ;
      =     M    125.2;
NETWORK
TITLE =

      L     DB1.DBD  464;
      L     L#0;
      <>D   ;
      =     M    125.3;
NETWORK
TITLE =

      L     DB1.DBD  404;
      L     L#0;
      <>D   ;
      =     M    125.4;
NETWORK
TITLE =

      L     DB1.DBD  424;
      L     L#0;
      <>D   ;
      =     M    125.5;
NETWORK
TITLE =

      L     DB1.DBD  444;
      L     L#0;
      <>D   ;
      =     M    125.6;
NETWORK
TITLE =

      L     DB101.DBD   64;
      L     L#0;
      ==D   ;
      =     M    126.0;
NETWORK
TITLE =

      L     DB1.DBD  364;
      L     L#0;
      ==D   ;
      =     M    126.1;
NETWORK
TITLE =
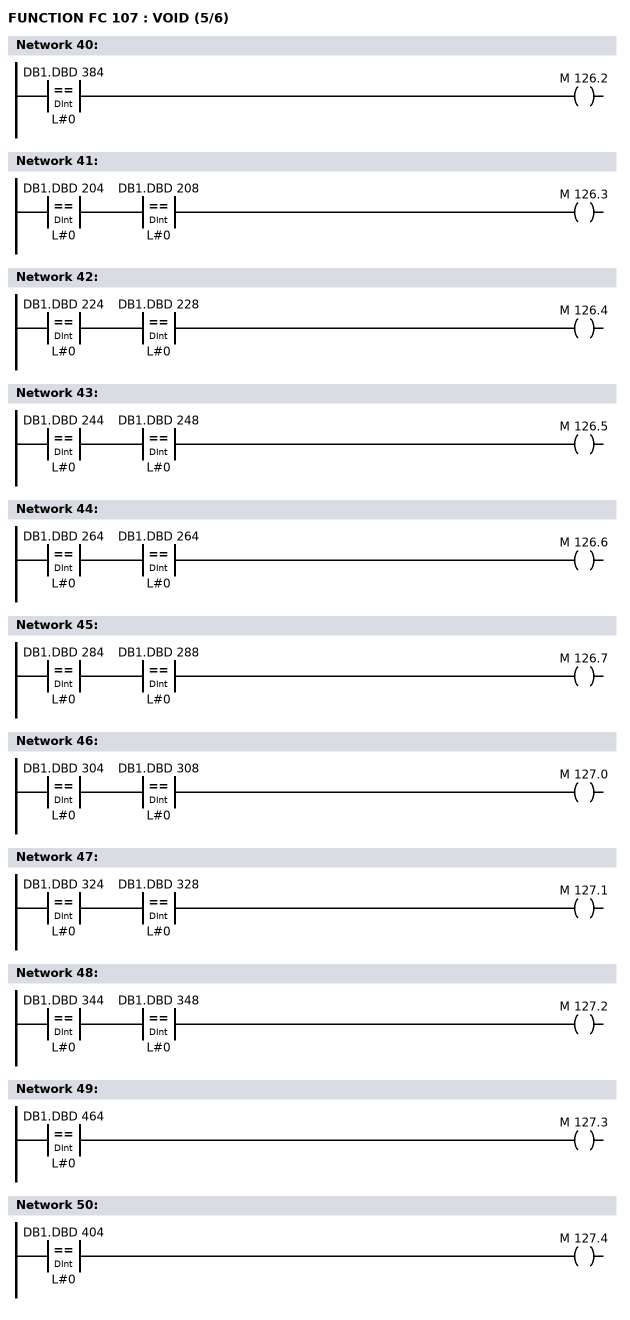

      L     DB1.DBD  384;
      L     L#0;
      ==D   ;
      =     M    126.2;
NETWORK
TITLE =

      A(    ;
      L     DB1.DBD  204;
      L     L#0;
      ==D   ;
      )     ;
      A(    ;
      L     DB1.DBD  208;
      L     L#0;
      ==D   ;
      )     ;
      =     M    126.3;
NETWORK
TITLE =

      A(    ;
      L     DB1.DBD  224;
      L     L#0;
      ==D   ;
      )     ;
      A(    ;
      L     DB1.DBD  228;
      L     L#0;
      ==D   ;
      )     ;
      =     M    126.4;
NETWORK
TITLE =

      A(    ;
      L     DB1.DBD  244;
      L     L#0;
      ==D   ;
      )     ;
      A(    ;
      L     DB1.DBD  248;
      L     L#0;
      ==D   ;
      )     ;
      =     M    126.5;
NETWORK
TITLE =

      A(    ;
      L     DB1.DBD  264;
      L     L#0;
      ==D   ;
      )     ;
      A(    ;
      L     DB1.DBD  264;
      L     L#0;
      ==D   ;
      )     ;
      =     M    126.6;
NETWORK
TITLE =

      A(    ;
      L     DB1.DBD  284;
      L     L#0;
      ==D   ;
      )     ;
      A(    ;
      L     DB1.DBD  288;
      L     L#0;
      ==D   ;
      )     ;
      =     M    126.7;
NETWORK
TITLE =

      A(    ;
      L     DB1.DBD  304;
      L     L#0;
      ==D   ;
      )     ;
      A(    ;
      L     DB1.DBD  308;
      L     L#0;
      ==D   ;
      )     ;
      =     M    127.0;
NETWORK
TITLE =

      A(    ;
      L     DB1.DBD  324;
      L     L#0;
      ==D   ;
      )     ;
      A(    ;
      L     DB1.DBD  328;
      L     L#0;
      ==D   ;
      )     ;
      =     M    127.1;
NETWORK
TITLE =

      A(    ;
      L     DB1.DBD  344;
      L     L#0;
      ==D   ;
      )     ;
      A(    ;
      L     DB1.DBD  348;
      L     L#0;
      ==D   ;
      )     ;
      =     M    127.2;
NETWORK
TITLE =

      L     DB1.DBD  464;
      L     L#0;
      ==D   ;
      =     M    127.3;
NETWORK
TITLE =

      L     DB1.DBD  404;
      L     L#0;
      ==D   ;
      =     M    127.4;
NETWORK
TITLE =
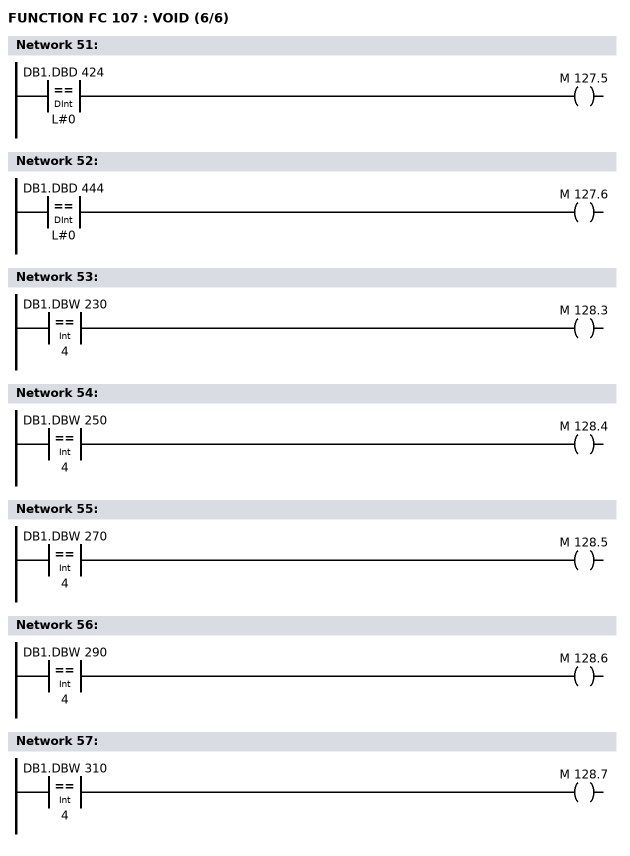

      L     DB1.DBD  424;
      L     L#0;
      ==D   ;
      =     M    127.5;
NETWORK
TITLE =

      L     DB1.DBD  444;
      L     L#0;
      ==D   ;
      =     M    127.6;
NETWORK
TITLE =

      L     DB1.DBW  230;
      L     4;
      ==I   ;
      =     M    128.3;
NETWORK
TITLE =

      L     DB1.DBW  250;
      L     4;
      ==I   ;
      =     M    128.4;
NETWORK
TITLE =

      L     DB1.DBW  270;
      L     4;
      ==I   ;
      =     M    128.5;
NETWORK
TITLE =

      L     DB1.DBW  290;
      L     4;
      ==I   ;
      =     M    128.6;
NETWORK
TITLE =

      L     DB1.DBW  310;
      L     4;
      ==I   ;
      =     M    128.7;
END_FUNCTION

FUNCTION_BLOCK FB 108
TITLE =
VERSION : 0.1

BEGIN
NETWORK
TITLE =PROFINET ERROR(1~10)
//
//
      A     M      3.3;
      =     L      0.0;
      A     L      0.0;
      A(    ;
      O     DB327.DBX 1025.3;
      O     ;
      A     M   7000.0;
      AN    I      0.1;
      AN    I    150.1;
      )     ;
      =     L      0.1;
      A     L      0.1;
      A     T    700;
      =     M   7000.0;
      A     L      0.1;
      BLD   102;
      L     S5T#0MS;
      SD    T    700;
      A     L      0.0;
      A(    ;
      O     DB327.DBX 1027.3;
      O     ;
      A     M   7000.1;
      AN    I      0.1;
      AN    I    150.1;
      )     ;
      =     L      0.1;
      A     L      0.1;
      A     T    701;
      =     M   7000.1;
      A     L      0.1;
      BLD   102;
      L     S5T#0MS;
      SD    T    701;
      A     L      0.0;
      A(    ;
      O     DB327.DBX 1029.3;
      O     ;
      A     M   7000.2;
      AN    I      0.1;
      AN    I    150.1;
      )     ;
      =     L      0.1;
      A     L      0.1;
      A     T    702;
      =     M   7000.2;
      A     L      0.1;
      BLD   102;
      L     S5T#0MS;
      SD    T    702;
      A     L      0.0;
      A(    ;
      O     DB327.DBX 1031.3;
      O     ;
      A     M   7000.3;
      AN    I      0.1;
      AN    I    150.1;
      )     ;
      =     L      0.1;
      A     L      0.1;
      A     T    703;
      =     M   7000.3;
      A     L      0.1;
      BLD   102;
      L     S5T#0MS;
      SD    T    703;
      A     L      0.0;
      A(    ;
      O     DB327.DBX 1033.3;
      O     ;
      A     M   7000.4;
      AN    I      0.1;
      AN    I    150.1;
      )     ;
      =     L      0.1;
      A     L      0.1;
      A     T    704;
      =     M   7000.4;
      A     L      0.1;
      BLD   102;
      L     S5T#0MS;
      SD    T    704;
      A     L      0.0;
      A(    ;
      O     DB327.DBX 1035.3;
      O     ;
      A     M   7000.5;
      AN    I      0.1;
      AN    I    150.1;
      )     ;
      =     L      0.1;
      A     L      0.1;
      A     T    705;
      =     M   7000.5;
      A     L      0.1;
      BLD   102;
      L     S5T#0MS;
      SD    T    705;
      A     L      0.0;
      A(    ;
      O     DB327.DBX 1037.3;
      O     ;
      A     M   7000.6;
      AN    I      0.1;
      AN    I    150.1;
      )     ;
      =     L      0.1;
      A     L      0.1;
      A     T    706;
      =     M   7000.6;
      A     L      0.1;
      BLD   102;
      L     S5T#0MS;
      SD    T    706;
      A     L      0.0;
      A(    ;
      O     DB327.DBX 1039.3;
      O     ;
      A     M   7000.7;
      AN    I      0.1;
      AN    I    150.1;
      )     ;
      =     L      0.1;
      A     L      0.1;
      A     T    707;
      =     M   7000.7;
      A     L      0.1;
      BLD   102;
      L     S5T#0MS;
      SD    T    707;
      A     L      0.0;
      A(    ;
      O     DB327.DBX 1041.3;
      O     ;
      A     M   7001.0;
      AN    I      0.1;
      AN    I    150.1;
      )     ;
      =     L      0.1;
      A     L      0.1;
      A     T    708;
      =     M   7001.0;
      A     L      0.1;
      BLD   102;
      L     S5T#0MS;
      SD    T    708;
      A     L      0.0;
      A(    ;
      O     DB327.DBX 1043.3;
      O     ;
      A     M   7001.1;
      AN    I      0.1;
      AN    I    150.1;
      )     ;
      =     L      0.1;
      A     L      0.1;
      A     T    709;
      =     M   7001.1;
      A     L      0.1;
      BLD   102;
      L     S5T#0MS;
      SD    T    709;
NETWORK
TITLE =PROFINET ERROR(11~20)
//
//
      A     M      3.3;
      =     L      0.0;
      A     L      0.0;
      A(    ;
      O     DB327.DBX 1045.3;
      O     ;
      A     M   7001.2;
      AN    I      0.1;
      AN    I    150.1;
      )     ;
      =     L      0.1;
      A     L      0.1;
      A     T    710;
      =     M   7001.2;
      A     L      0.1;
      BLD   102;
      L     S5T#0MS;
      SD    T    710;
      A     L      0.0;
      A(    ;
      O     DB327.DBX 1047.3;
      O     ;
      A     M   7001.3;
      AN    I      0.1;
      AN    I    150.1;
      )     ;
      =     L      0.1;
      A     L      0.1;
      A     T    711;
      =     M   7001.3;
      A     L      0.1;
      BLD   102;
      L     S5T#0MS;
      SD    T    711;
      A     L      0.0;
      A(    ;
      O     DB327.DBX 1049.3;
      O     ;
      A     M   7001.4;
      AN    I      0.1;
      AN    I    150.1;
      )     ;
      =     L      0.1;
      A     L      0.1;
      A     T    712;
      =     M   7001.4;
      A     L      0.1;
      BLD   102;
      L     S5T#0MS;
      SD    T    712;
      A     L      0.0;
      A(    ;
      O     DB327.DBX 1051.3;
      O     ;
      A     M   7001.5;
      AN    I      0.1;
      AN    I    150.1;
      )     ;
      =     L      0.1;
      A     L      0.1;
      A     T    713;
      =     M   7001.5;
      A     L      0.1;
      BLD   102;
      L     S5T#0MS;
      SD    T    713;
      A     L      0.0;
      A(    ;
      O     DB327.DBX 1053.3;
      O     ;
      A     M   7001.6;
      AN    I      0.1;
      AN    I    150.1;
      )     ;
      =     L      0.1;
      A     L      0.1;
      A     T    714;
      =     M   7001.6;
      A     L      0.1;
      BLD   102;
      L     S5T#0MS;
      SD    T    714;
      A     L      0.0;
      A(    ;
      O     DB327.DBX 1055.3;
      O     ;
      A     M   7001.7;
      AN    I      0.1;
      AN    I    150.1;
      )     ;
      =     L      0.1;
      A     L      0.1;
      A     T    715;
      =     M   7001.7;
      A     L      0.1;
      BLD   102;
      L     S5T#0MS;
      SD    T    715;
      A     L      0.0;
      A(    ;
      O     DB327.DBX 1057.3;
      O     ;
      A     M   7002.0;
      AN    I      0.1;
      AN    I    150.1;
      )     ;
      =     L      0.1;
      A     L      0.1;
      A     T    716;
      =     M   7002.0;
      A     L      0.1;
      BLD   102;
      L     S5T#0MS;
      SD    T    716;
      A     L      0.0;
      A(    ;
      O     DB327.DBX 1059.3;
      O     ;
      A     M   7002.1;
      AN    I      0.1;
      AN    I    150.1;
      )     ;
      =     L      0.1;
      A     L      0.1;
      A     T    717;
      =     M   7002.1;
      A     L      0.1;
      BLD   102;
      L     S5T#0MS;
      SD    T    717;
      A     L      0.0;
      A(    ;
      O     DB327.DBX 1061.3;
      O     ;
      A     M   7002.2;
      AN    I      0.1;
      AN    I    150.1;
      )     ;
      =     L      0.1;
      A     L      0.1;
      A     T    718;
      =     M   7002.2;
      A     L      0.1;
      BLD   102;
      L     S5T#0MS;
      SD    T    718;
      A     L      0.0;
      A(    ;
      O     DB327.DBX 1063.3;
      O     ;
      A     M   7002.3;
      AN    I      0.1;
      AN    I    150.1;
      )     ;
      =     L      0.1;
      A     L      0.1;
      A     T    719;
      =     M   7002.3;
      A     L      0.1;
      BLD   102;
      L     S5T#0MS;
      SD    T    719;
NETWORK
TITLE =PROFINET ERROR(21~30)
//
//
      A     M      3.3;
      =     L      0.0;
      A     L      0.0;
      A(    ;
      O     DB327.DBX 1065.3;
      O     ;
      A     M   7002.4;
      AN    I      0.1;
      AN    I    150.1;
      )     ;
      =     L      0.1;
      A     L      0.1;
      A     T    720;
      =     M   7002.4;
      A     L      0.1;
      BLD   102;
      L     S5T#0MS;
      SD    T    720;
      A     L      0.0;
      A(    ;
      O     DB327.DBX 1067.3;
      O     ;
      A     M   7002.5;
      AN    I      0.1;
      AN    I    150.1;
      )     ;
      =     L      0.1;
      A     L      0.1;
      A     T    721;
      =     M   7002.5;
      A     L      0.1;
      BLD   102;
      L     S5T#0MS;
      SD    T    721;
      A     L      0.0;
      A(    ;
      O     DB327.DBX 1069.3;
      O     ;
      A     M   7002.6;
      AN    I      0.1;
      AN    I    150.1;
      )     ;
      =     L      0.1;
      A     L      0.1;
      A     T    722;
      =     M   7002.6;
      A     L      0.1;
      BLD   102;
      L     S5T#0MS;
      SD    T    722;
      A     L      0.0;
      A(    ;
      O     DB327.DBX 1071.3;
      O     ;
      A     M   7002.7;
      AN    I      0.1;
      AN    I    150.1;
      )     ;
      =     L      0.1;
      A     L      0.1;
      A     T    723;
      =     M   7002.7;
      A     L      0.1;
      BLD   102;
      L     S5T#0MS;
      SD    T    723;
      A     L      0.0;
      A(    ;
      O     DB327.DBX 1073.3;
      O     ;
      A     M   7003.0;
      AN    I      0.1;
      AN    I    150.1;
      )     ;
      =     L      0.1;
      A     L      0.1;
      A     T    724;
      =     M   7003.0;
      A     L      0.1;
      BLD   102;
      L     S5T#0MS;
      SD    T    724;
      A     L      0.0;
      A(    ;
      O     DB327.DBX 1075.3;
      O     ;
      A     M   7003.1;
      AN    I      0.1;
      AN    I    150.1;
      )     ;
      =     L      0.1;
      A     L      0.1;
      A     T    725;
      AN    M      3.3;
      =     M   7003.1;
      A     L      0.1;
      BLD   102;
      L     S5T#0MS;
      SD    T    725;
      A     L      0.0;
      A(    ;
      O     DB327.DBX 1077.3;
      O     ;
      A     M   7003.2;
      AN    I      0.1;
      AN    I    150.1;
      )     ;
      =     L      0.1;
      A     L      0.1;
      A     T    726;
      AN    M      3.3;
      =     M   7003.2;
      A     L      0.1;
      BLD   102;
      L     S5T#0MS;
      SD    T    726;
      A     L      0.0;
      A(    ;
      O     DB327.DBX 1079.3;
      O     ;
      A     M   7003.3;
      AN    I      0.1;
      AN    I    150.1;
      )     ;
      =     L      0.1;
      A     L      0.1;
      A     T    727;
      AN    M      3.3;
      =     M   7003.3;
      A     L      0.1;
      BLD   102;
      L     S5T#0MS;
      SD    T    727;
      A     L      0.0;
      A(    ;
      O     DB327.DBX 1081.3;
      O     ;
      A     M   7003.4;
      AN    I      0.1;
      AN    I    150.1;
      )     ;
      =     L      0.1;
      A     L      0.1;
      A     T    728;
      AN    M      3.3;
      =     M   7003.4;
      A     L      0.1;
      BLD   102;
      L     S5T#0MS;
      SD    T    728;
      A     L      0.0;
      A(    ;
      O     DB327.DBX 1083.3;
      O     ;
      A     M   7003.5;
      AN    I      0.1;
      AN    I    150.1;
      )     ;
      =     L      0.1;
      A     L      0.1;
      A     T    729;
      AN    M      3.3;
      =     M   7003.5;
      A     L      0.1;
      BLD   102;
      L     S5T#0MS;
      SD    T    729;
NETWORK
TITLE =PROFINET ERROR(31~40)
//
//
      A     M      3.3;
      =     L      0.0;
      A     L      0.0;
      A(    ;
      O     DB327.DBX 1085.3;
      O     ;
      A     M   7003.6;
      AN    I      0.1;
      AN    I    150.1;
      )     ;
      =     L      0.1;
      A     L      0.1;
      A     T    730;
      AN    M      3.3;
      =     M   7003.6;
      A     L      0.1;
      BLD   102;
      L     S5T#0MS;
      SD    T    730;
      A     L      0.0;
      A(    ;
      O     DB327.DBX 1087.3;
      O     ;
      A     M   7003.7;
      AN    I      0.1;
      AN    I    150.1;
      )     ;
      =     L      0.1;
      A     L      0.1;
      A     T    731;
      AN    M      3.3;
      =     M   7003.7;
      A     L      0.1;
      BLD   102;
      L     S5T#0MS;
      SD    T    731;
      A     L      0.0;
      A(    ;
      O     DB327.DBX 1089.3;
      O     ;
      A     M   7004.0;
      AN    I      0.1;
      AN    I    150.1;
      )     ;
      =     L      0.1;
      A     L      0.1;
      A     T    732;
      AN    M      3.3;
      =     M   7004.0;
      A     L      0.1;
      BLD   102;
      L     S5T#0MS;
      SD    T    732;
      A     L      0.0;
      A(    ;
      O     DB327.DBX 1091.3;
      O     ;
      A     M   7004.1;
      AN    I      0.1;
      AN    I    150.1;
      )     ;
      =     L      0.1;
      A     L      0.1;
      A     T    733;
      AN    M      3.3;
      =     M   7004.1;
      A     L      0.1;
      BLD   102;
      L     S5T#0MS;
      SD    T    733;
      A     L      0.0;
      A(    ;
      O     DB327.DBX 1093.3;
      O     ;
      A     M   7004.2;
      AN    I      0.1;
      AN    I    150.1;
      )     ;
      =     L      0.1;
      A     L      0.1;
      A     T    734;
      AN    M      3.3;
      =     M   7004.2;
      A     L      0.1;
      BLD   102;
      L     S5T#0MS;
      SD    T    734;
      A     L      0.0;
      A(    ;
      O     DB327.DBX 1095.3;
      O     ;
      A     M   7004.3;
      AN    I      0.1;
      AN    I    150.1;
      )     ;
      =     L      0.1;
      A     L      0.1;
      A     T    735;
      AN    M      3.3;
      =     M   7004.3;
      A     L      0.1;
      BLD   102;
      L     S5T#0MS;
      SD    T    735;
      A     L      0.0;
      A(    ;
      O     DB327.DBX 1097.3;
      O     ;
      A     M   7004.4;
      AN    I      0.1;
      AN    I    150.1;
      )     ;
      =     L      0.1;
      A     L      0.1;
      A     T    736;
      AN    M      3.3;
      =     M   7004.4;
      A     L      0.1;
      BLD   102;
      L     S5T#0MS;
      SD    T    736;
      A     L      0.0;
      A(    ;
      O     DB327.DBX 1099.3;
      O     ;
      A     M   7004.5;
      AN    I      0.1;
      AN    I    150.1;
      )     ;
      =     L      0.1;
      A     L      0.1;
      A     T    737;
      AN    M      3.3;
      =     M   7004.5;
      A     L      0.1;
      BLD   102;
      L     S5T#0MS;
      SD    T    737;
      A     L      0.0;
      A(    ;
      O     DB327.DBX 1101.3;
      O     ;
      A     M   7004.6;
      AN    I      0.1;
      AN    I    150.1;
      )     ;
      =     L      0.1;
      A     L      0.1;
      A     T    738;
      AN    M      3.3;
      =     M   7004.6;
      A     L      0.1;
      BLD   102;
      L     S5T#0MS;
      SD    T    738;
      A     L      0.0;
      A(    ;
      O     DB327.DBX 1103.3;
      O     ;
      A     M   7004.7;
      AN    I      0.1;
      AN    I    150.1;
      )     ;
      =     L      0.1;
      A     L      0.1;
      A     T    739;
      AN    M      3.3;
      =     M   7004.7;
      A     L      0.1;
      BLD   102;
      L     S5T#0MS;
      SD    T    739;
NETWORK
TITLE =PROFINET ERROR(150~159)

      A     M      3.3;
      =     L      0.0;
      A     L      0.0;
      A(    ;
      O     DB327.DBX 1323.3;
      O     ;
      A     M   7018.5;
      AN    I      0.1;
      AN    I    150.1;
      )     ;
      =     L      0.1;
      A     L      0.1;
      A     T    849;
      =     M   7018.5;
      A     L      0.1;
      BLD   102;
      L     S5T#0MS;
      SD    T    849;
      A     L      0.0;
      A(    ;
      O     DB327.DBX 1325.3;
      O     ;
      A     M   7018.6;
      AN    I      0.1;
      AN    I    150.1;
      )     ;
      =     L      0.1;
      A     L      0.1;
      A     T    850;
      =     M   7018.6;
      A     L      0.1;
      BLD   102;
      L     S5T#0MS;
      SD    T    850;
      A     L      0.0;
      A(    ;
      O     DB327.DBX 1327.3;
      O     ;
      A     M   7018.7;
      AN    I      0.1;
      AN    I    150.1;
      )     ;
      =     L      0.1;
      A     L      0.1;
      A     T    851;
      AN    M      3.3;
      =     M   7018.7;
      A     L      0.1;
      BLD   102;
      L     S5T#0MS;
      SD    T    851;
      A     L      0.0;
      A(    ;
      O     DB327.DBX 1329.3;
      O     ;
      A     M   7019.0;
      AN    I      0.1;
      AN    I    150.1;
      )     ;
      =     L      0.1;
      A     L      0.1;
      A     T    852;
      AN    M      3.3;
      =     M   7019.0;
      A     L      0.1;
      BLD   102;
      L     S5T#0MS;
      SD    T    852;
      A     L      0.0;
      A(    ;
      O     DB327.DBX 1331.3;
      O     ;
      A     M   7019.1;
      AN    I      0.1;
      AN    I    150.1;
      )     ;
      =     L      0.1;
      A     L      0.1;
      A     T    853;
      AN    M      3.3;
      =     M   7019.1;
      A     L      0.1;
      BLD   102;
      L     S5T#0MS;
      SD    T    853;
      A     L      0.0;
      A(    ;
      O     DB327.DBX 1333.3;
      O     ;
      A     M   7019.2;
      AN    I      0.1;
      AN    I    150.1;
      )     ;
      =     L      0.1;
      A     L      0.1;
      A     T    854;
      AN    M      3.3;
      =     M   7019.2;
      A     L      0.1;
      BLD   102;
      L     S5T#0MS;
      SD    T    854;
      A     L      0.0;
      A(    ;
      O     DB327.DBX 1335.3;
      O     ;
      A     M   7019.3;
      AN    I      0.1;
      AN    I    150.1;
      )     ;
      =     L      0.1;
      A     L      0.1;
      A     T    855;
      AN    M      3.3;
      =     M   7019.3;
      A     L      0.1;
      BLD   102;
      L     S5T#0MS;
      SD    T    855;
      A     L      0.0;
      A(    ;
      O     DB327.DBX 1337.3;
      O     ;
      A     M   7019.4;
      AN    I      0.1;
      AN    I    150.1;
      )     ;
      =     L      0.1;
      A     L      0.1;
      A     T    856;
      AN    M      3.3;
      =     M   7019.4;
      A     L      0.1;
      BLD   102;
      L     S5T#0MS;
      SD    T    856;
      A     L      0.0;
      A(    ;
      O     DB327.DBX 1339.3;
      O     ;
      A     M   7019.5;
      AN    I      0.1;
      AN    I    150.1;
      )     ;
      =     L      0.1;
      A     L      0.1;
      A     T    857;
      AN    M      3.3;
      =     M   7019.5;
      A     L      0.1;
      BLD   102;
      L     S5T#0MS;
      SD    T    857;
      A     L      0.0;
      A(    ;
      O     DB327.DBX 1341.3;
      O     ;
      A     M   7019.6;
      AN    I      0.1;
      AN    I    150.1;
      )     ;
      =     L      0.1;
      A     L      0.1;
      A     T    858;
      AN    M      3.3;
      =     M   7019.6;
      A     L      0.1;
      BLD   102;
      L     S5T#0MS;
      SD    T    858;
NETWORK
TITLE =CP TRIP(20~29)
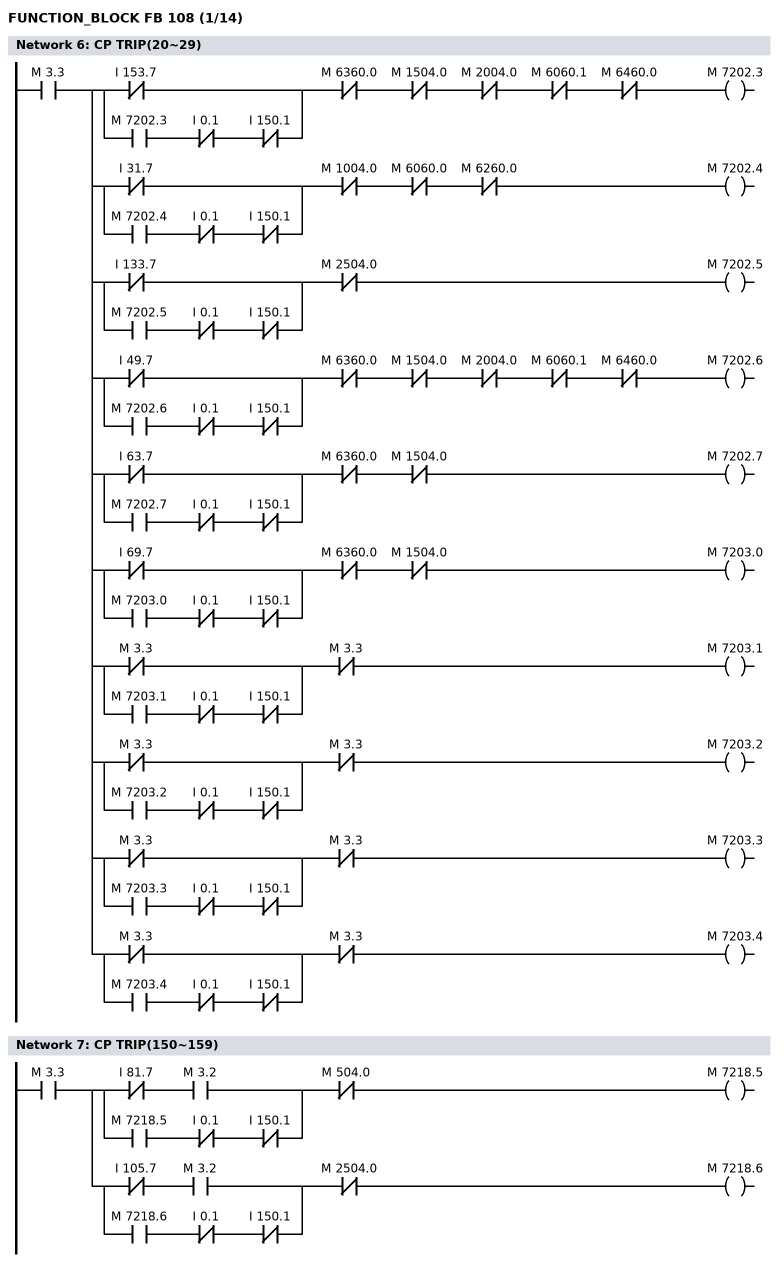

      A     M      3.3;
      =     L      0.0;
      A     L      0.0;
      A(    ;
      ON    I    153.7;
      O     ;
      A     M   7202.3;
      AN    I      0.1;
      AN    I    150.1;
      )     ;
      AN    M   6360.0;
      AN    M   1504.0;
      AN    M   2004.0;
      AN    M   6060.1;
      AN    M   6460.0;
      =     M   7202.3;
      A     L      0.0;
      A(    ;
      ON    I     31.7;
      O     ;
      A     M   7202.4;
      AN    I      0.1;
      AN    I    150.1;
      )     ;
      AN    M   1004.0;
      AN    M   6060.0;
      AN    M   6260.0;
      =     M   7202.4;
      A     L      0.0;
      A(    ;
      ON    I    133.7;
      O     ;
      A     M   7202.5;
      AN    I      0.1;
      AN    I    150.1;
      )     ;
      AN    M   2504.0;
      =     M   7202.5;
      A     L      0.0;
      A(    ;
      ON    I     49.7;
      O     ;
      A     M   7202.6;
      AN    I      0.1;
      AN    I    150.1;
      )     ;
      AN    M   6360.0;
      AN    M   1504.0;
      AN    M   2004.0;
      AN    M   6060.1;
      AN    M   6460.0;
      =     M   7202.6;
      A     L      0.0;
      A(    ;
      ON    I     63.7;
      O     ;
      A     M   7202.7;
      AN    I      0.1;
      AN    I    150.1;
      )     ;
      AN    M   6360.0;
      AN    M   1504.0;
      =     M   7202.7;
      A     L      0.0;
      A(    ;
      ON    I     69.7;
      O     ;
      A     M   7203.0;
      AN    I      0.1;
      AN    I    150.1;
      )     ;
      AN    M   6360.0;
      AN    M   1504.0;
      =     M   7203.0;
      A     L      0.0;
      A(    ;
      ON    M      3.3;
      O     ;
      A     M   7203.1;
      AN    I      0.1;
      AN    I    150.1;
      )     ;
      AN    M      3.3;
      =     M   7203.1;
      A     L      0.0;
      A(    ;
      ON    M      3.3;
      O     ;
      A     M   7203.2;
      AN    I      0.1;
      AN    I    150.1;
      )     ;
      AN    M      3.3;
      =     M   7203.2;
      A     L      0.0;
      A(    ;
      ON    M      3.3;
      O     ;
      A     M   7203.3;
      AN    I      0.1;
      AN    I    150.1;
      )     ;
      AN    M      3.3;
      =     M   7203.3;
      A     L      0.0;
      A(    ;
      ON    M      3.3;
      O     ;
      A     M   7203.4;
      AN    I      0.1;
      AN    I    150.1;
      )     ;
      AN    M      3.3;
      =     M   7203.4;
NETWORK
TITLE =CP TRIP(150~159)

      A     M      3.3;
      =     L      0.0;
      A     L      0.0;
      A(    ;
      AN    I     81.7;
      A     M      3.2;
      O     ;
      A     M   7218.5;
      AN    I      0.1;
      AN    I    150.1;
      )     ;
      AN    M    504.0;
      =     M   7218.5;
      A     L      0.0;
      A(    ;
      AN    I    105.7;
      A     M      3.2;
      O     ;
      A     M   7218.6;
      AN    I      0.1;
      AN    I    150.1;
      )     ;
      AN    M   2504.0;
      =     M   7218.6;
NETWORK
TITLE =통신확인 비트(M5159.7) 1초 플리커
//
//
//
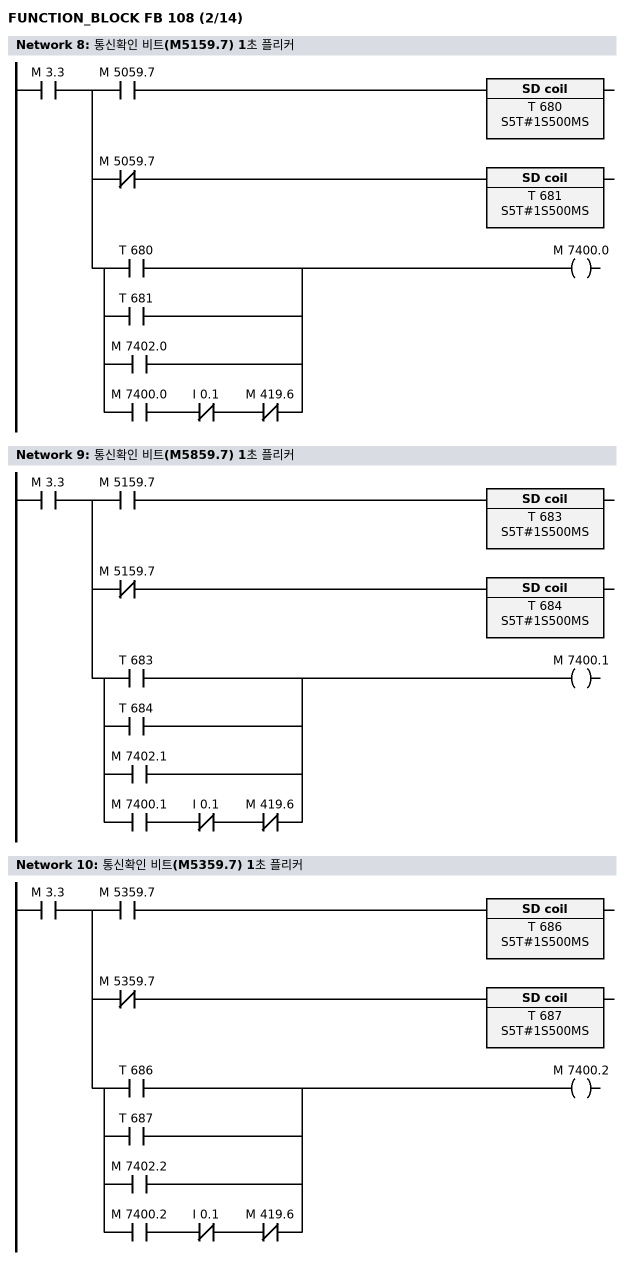
      A     M      3.3;
      =     L      0.0;
      A     L      0.0;
      A     M   5059.7;
      L     S5T#1S500MS;
      SD    T    680;
      A     L      0.0;
      AN    M   5059.7;
      L     S5T#1S500MS;
      SD    T    681;
      A     L      0.0;
      A(    ;
      O     T    680;
      O     T    681;
      O     M   7402.0;
      O     ;
      A     M   7400.0;
      AN    I      0.1;
      AN    M    419.6;
      )     ;
      =     M   7400.0;
NETWORK
TITLE =통신확인 비트(M5859.7) 1초 플리커
//
//
//
      A     M      3.3;
      =     L      0.0;
      A     L      0.0;
      A     M   5159.7;
      L     S5T#1S500MS;
      SD    T    683;
      A     L      0.0;
      AN    M   5159.7;
      L     S5T#1S500MS;
      SD    T    684;
      A     L      0.0;
      A(    ;
      O     T    683;
      O     T    684;
      O     M   7402.1;
      O     ;
      A     M   7400.1;
      AN    I      0.1;
      AN    M    419.6;
      )     ;
      =     M   7400.1;
NETWORK
TITLE =통신확인 비트(M5359.7) 1초 플리커
//
//
//
      A     M      3.3;
      =     L      0.0;
      A     L      0.0;
      A     M   5359.7;
      L     S5T#1S500MS;
      SD    T    686;
      A     L      0.0;
      AN    M   5359.7;
      L     S5T#1S500MS;
      SD    T    687;
      A     L      0.0;
      A(    ;
      O     T    686;
      O     T    687;
      O     M   7402.2;
      O     ;
      A     M   7400.2;
      AN    I      0.1;
      AN    M    419.6;
      )     ;
      =     M   7400.2;
NETWORK
TITLE =통신확인 비트(M5459.7) 1초 플리커
//
//
//
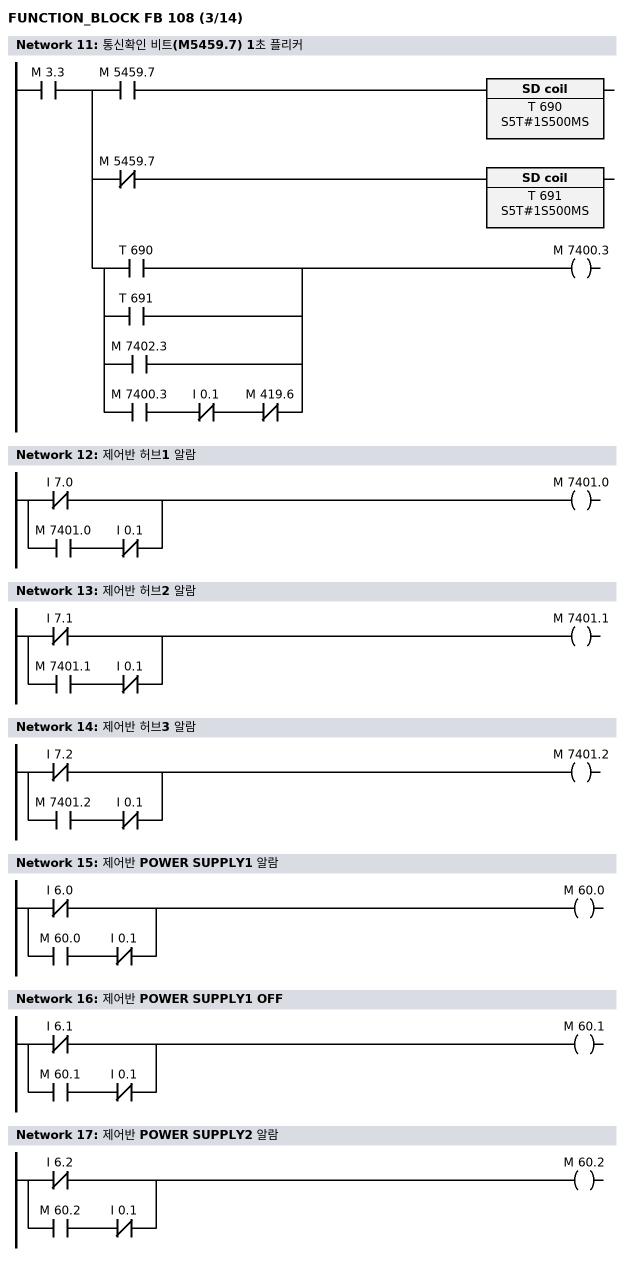
      A     M      3.3;
      =     L      0.0;
      A     L      0.0;
      A     M   5459.7;
      L     S5T#1S500MS;
      SD    T    690;
      A     L      0.0;
      AN    M   5459.7;
      L     S5T#1S500MS;
      SD    T    691;
      A     L      0.0;
      A(    ;
      O     T    690;
      O     T    691;
      O     M   7402.3;
      O     ;
      A     M   7400.3;
      AN    I      0.1;
      AN    M    419.6;
      )     ;
      =     M   7400.3;
NETWORK
TITLE =제어반 허브1 알람

      ON    I      7.0;
      O     ;
      A     M   7401.0;
      AN    I      0.1;
      =     M   7401.0;
NETWORK
TITLE =제어반 허브2 알람

      ON    I      7.1;
      O     ;
      A     M   7401.1;
      AN    I      0.1;
      =     M   7401.1;
NETWORK
TITLE =제어반 허브3 알람

      ON    I      7.2;
      O     ;
      A     M   7401.2;
      AN    I      0.1;
      =     M   7401.2;
NETWORK
TITLE =제어반 POWER SUPPLY1 알람

      ON    I      6.0;
      O     ;
      A     M     60.0;
      AN    I      0.1;
      =     M     60.0;
NETWORK
TITLE =제어반 POWER SUPPLY1 OFF

      ON    I      6.1;
      O     ;
      A     M     60.1;
      AN    I      0.1;
      =     M     60.1;
NETWORK
TITLE =제어반 POWER SUPPLY2 알람
//
//
      ON    I      6.2;
      O     ;
      A     M     60.2;
      AN    I      0.1;
      =     M     60.2;
NETWORK
TITLE =제어반 POWER SUPPLY2 OFF
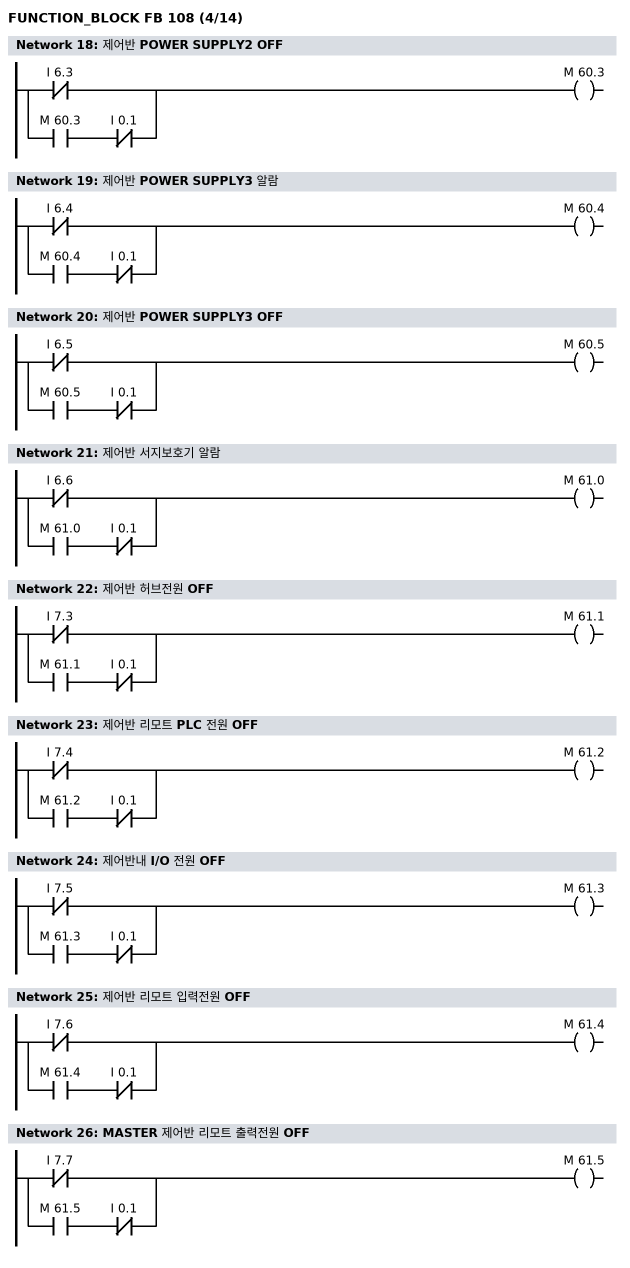

      ON    I      6.3;
      O     ;
      A     M     60.3;
      AN    I      0.1;
      =     M     60.3;
NETWORK
TITLE =제어반 POWER SUPPLY3 알람
//
//
      ON    I      6.4;
      O     ;
      A     M     60.4;
      AN    I      0.1;
      =     M     60.4;
NETWORK
TITLE =제어반 POWER SUPPLY3 OFF

      ON    I      6.5;
      O     ;
      A     M     60.5;
      AN    I      0.1;
      =     M     60.5;
NETWORK
TITLE =제어반 서지보호기 알람

      ON    I      6.6;
      O     ;
      A     M     61.0;
      AN    I      0.1;
      =     M     61.0;
NETWORK
TITLE =제어반 허브전원 OFF

      ON    I      7.3;
      O     ;
      A     M     61.1;
      AN    I      0.1;
      =     M     61.1;
NETWORK
TITLE =제어반 리모트 PLC 전원 OFF

      ON    I      7.4;
      O     ;
      A     M     61.2;
      AN    I      0.1;
      =     M     61.2;
NETWORK
TITLE =제어반내 I/O 전원 OFF

      ON    I      7.5;
      O     ;
      A     M     61.3;
      AN    I      0.1;
      =     M     61.3;
NETWORK
TITLE =제어반 리모트 입력전원 OFF

      ON    I      7.6;
      O     ;
      A     M     61.4;
      AN    I      0.1;
      =     M     61.4;
NETWORK
TITLE =MASTER 제어반 리모트 출력전원 OFF

      ON    I      7.7;
      O     ;
      A     M     61.5;
      AN    I      0.1;
      =     M     61.5;
NETWORK
TITLE =PROFINET ALARM-모듈이상이나 통신케이블단선(1~10)
//
//
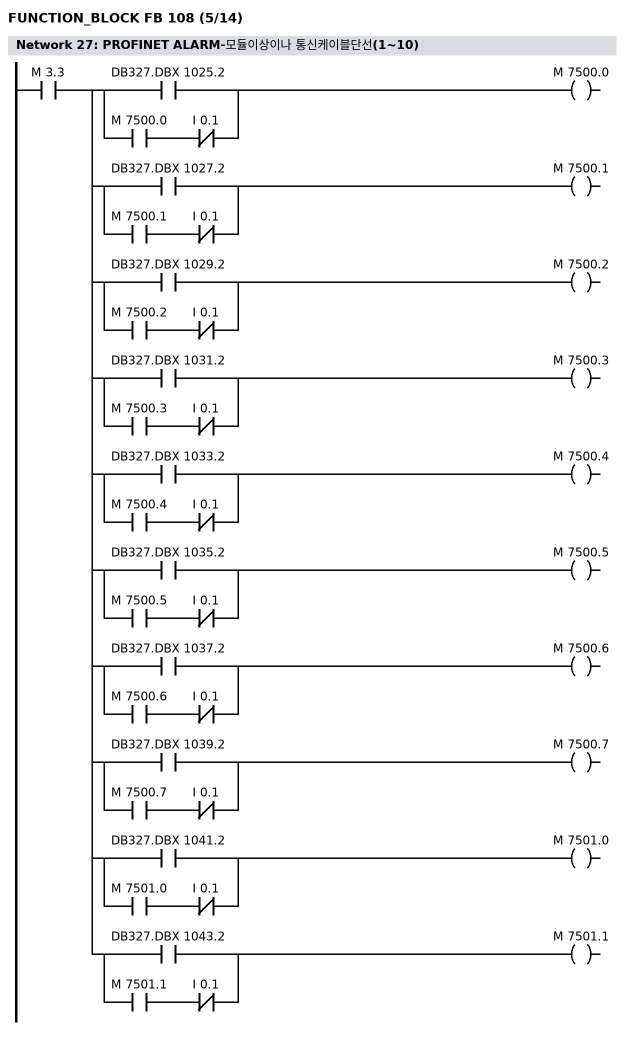
      A     M      3.3;
      =     L      0.0;
      A     L      0.0;
      A(    ;
      O     DB327.DBX 1025.2;
      O     ;
      A     M   7500.0;
      AN    I      0.1;
      )     ;
      =     M   7500.0;
      A     L      0.0;
      A(    ;
      O     DB327.DBX 1027.2;
      O     ;
      A     M   7500.1;
      AN    I      0.1;
      )     ;
      =     M   7500.1;
      A     L      0.0;
      A(    ;
      O     DB327.DBX 1029.2;
      O     ;
      A     M   7500.2;
      AN    I      0.1;
      )     ;
      =     M   7500.2;
      A     L      0.0;
      A(    ;
      O     DB327.DBX 1031.2;
      O     ;
      A     M   7500.3;
      AN    I      0.1;
      )     ;
      =     M   7500.3;
      A     L      0.0;
      A(    ;
      O     DB327.DBX 1033.2;
      O     ;
      A     M   7500.4;
      AN    I      0.1;
      )     ;
      =     M   7500.4;
      A     L      0.0;
      A(    ;
      O     DB327.DBX 1035.2;
      O     ;
      A     M   7500.5;
      AN    I      0.1;
      )     ;
      =     M   7500.5;
      A     L      0.0;
      A(    ;
      O     DB327.DBX 1037.2;
      O     ;
      A     M   7500.6;
      AN    I      0.1;
      )     ;
      =     M   7500.6;
      A     L      0.0;
      A(    ;
      O     DB327.DBX 1039.2;
      O     ;
      A     M   7500.7;
      AN    I      0.1;
      )     ;
      =     M   7500.7;
      A     L      0.0;
      A(    ;
      O     DB327.DBX 1041.2;
      O     ;
      A     M   7501.0;
      AN    I      0.1;
      )     ;
      =     M   7501.0;
      A     L      0.0;
      A(    ;
      O     DB327.DBX 1043.2;
      O     ;
      A     M   7501.1;
      AN    I      0.1;
      )     ;
      =     M   7501.1;
NETWORK
TITLE =PROFINET ALARM-모듈이상이나 통신케이블단선(11~20)
//
//
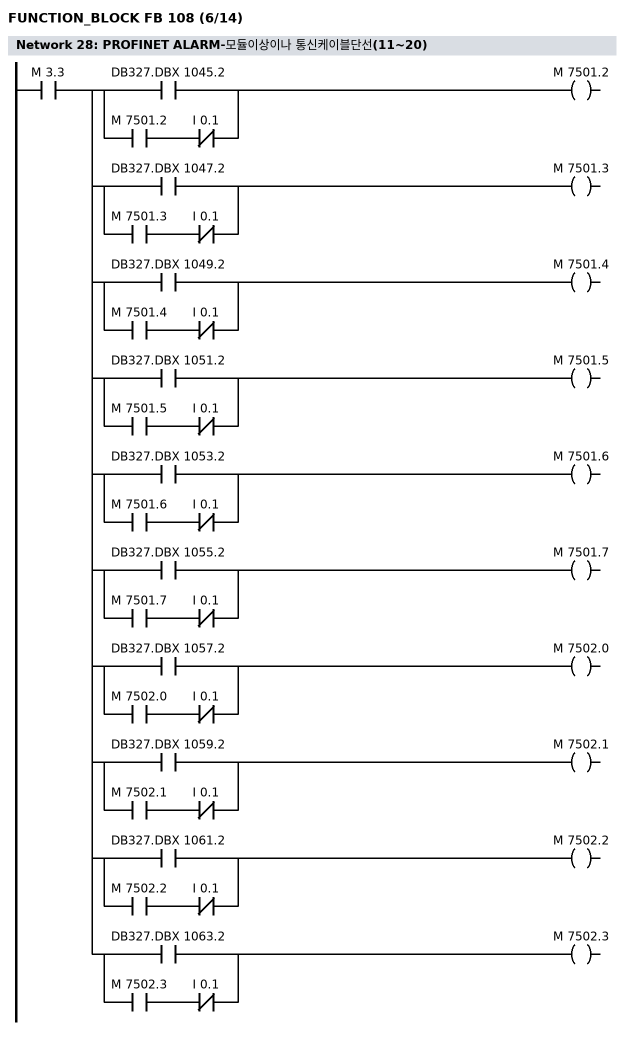
      A     M      3.3;
      =     L      0.0;
      A     L      0.0;
      A(    ;
      O     DB327.DBX 1045.2;
      O     ;
      A     M   7501.2;
      AN    I      0.1;
      )     ;
      =     M   7501.2;
      A     L      0.0;
      A(    ;
      O     DB327.DBX 1047.2;
      O     ;
      A     M   7501.3;
      AN    I      0.1;
      )     ;
      =     M   7501.3;
      A     L      0.0;
      A(    ;
      O     DB327.DBX 1049.2;
      O     ;
      A     M   7501.4;
      AN    I      0.1;
      )     ;
      =     M   7501.4;
      A     L      0.0;
      A(    ;
      O     DB327.DBX 1051.2;
      O     ;
      A     M   7501.5;
      AN    I      0.1;
      )     ;
      =     M   7501.5;
      A     L      0.0;
      A(    ;
      O     DB327.DBX 1053.2;
      O     ;
      A     M   7501.6;
      AN    I      0.1;
      )     ;
      =     M   7501.6;
      A     L      0.0;
      A(    ;
      O     DB327.DBX 1055.2;
      O     ;
      A     M   7501.7;
      AN    I      0.1;
      )     ;
      =     M   7501.7;
      A     L      0.0;
      A(    ;
      O     DB327.DBX 1057.2;
      O     ;
      A     M   7502.0;
      AN    I      0.1;
      )     ;
      =     M   7502.0;
      A     L      0.0;
      A(    ;
      O     DB327.DBX 1059.2;
      O     ;
      A     M   7502.1;
      AN    I      0.1;
      )     ;
      =     M   7502.1;
      A     L      0.0;
      A(    ;
      O     DB327.DBX 1061.2;
      O     ;
      A     M   7502.2;
      AN    I      0.1;
      )     ;
      =     M   7502.2;
      A     L      0.0;
      A(    ;
      O     DB327.DBX 1063.2;
      O     ;
      A     M   7502.3;
      AN    I      0.1;
      )     ;
      =     M   7502.3;
NETWORK
TITLE =PROFINET ALARM-모듈이상이나 통신케이블단선(21~30)
//
//
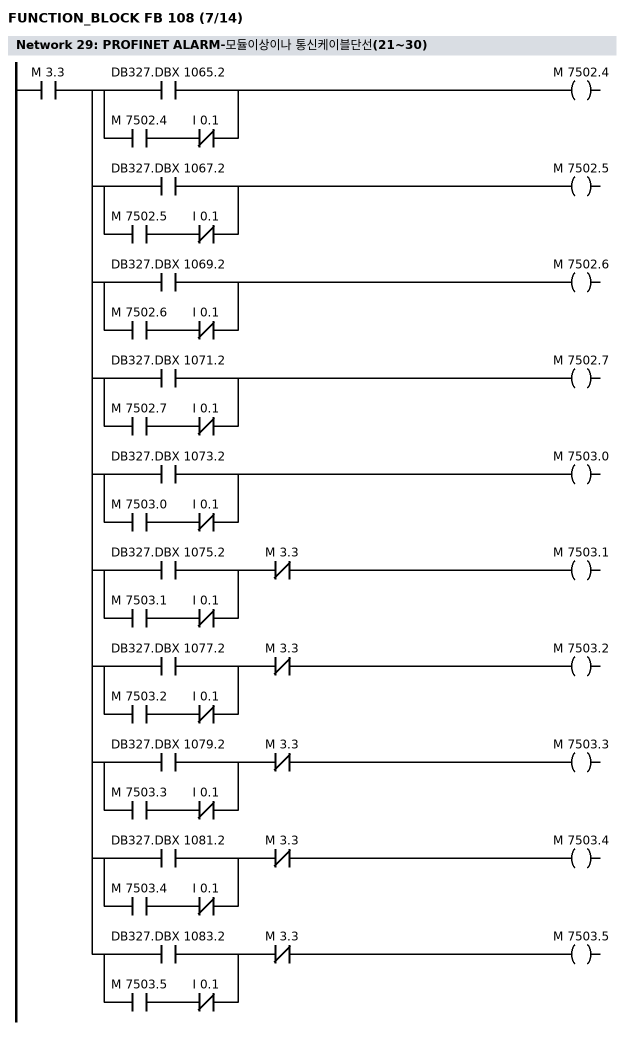
      A     M      3.3;
      =     L      0.0;
      A     L      0.0;
      A(    ;
      O     DB327.DBX 1065.2;
      O     ;
      A     M   7502.4;
      AN    I      0.1;
      )     ;
      =     M   7502.4;
      A     L      0.0;
      A(    ;
      O     DB327.DBX 1067.2;
      O     ;
      A     M   7502.5;
      AN    I      0.1;
      )     ;
      =     M   7502.5;
      A     L      0.0;
      A(    ;
      O     DB327.DBX 1069.2;
      O     ;
      A     M   7502.6;
      AN    I      0.1;
      )     ;
      =     M   7502.6;
      A     L      0.0;
      A(    ;
      O     DB327.DBX 1071.2;
      O     ;
      A     M   7502.7;
      AN    I      0.1;
      )     ;
      =     M   7502.7;
      A     L      0.0;
      A(    ;
      O     DB327.DBX 1073.2;
      O     ;
      A     M   7503.0;
      AN    I      0.1;
      )     ;
      =     M   7503.0;
      A     L      0.0;
      A(    ;
      O     DB327.DBX 1075.2;
      O     ;
      A     M   7503.1;
      AN    I      0.1;
      )     ;
      AN    M      3.3;
      =     M   7503.1;
      A     L      0.0;
      A(    ;
      O     DB327.DBX 1077.2;
      O     ;
      A     M   7503.2;
      AN    I      0.1;
      )     ;
      AN    M      3.3;
      =     M   7503.2;
      A     L      0.0;
      A(    ;
      O     DB327.DBX 1079.2;
      O     ;
      A     M   7503.3;
      AN    I      0.1;
      )     ;
      AN    M      3.3;
      =     M   7503.3;
      A     L      0.0;
      A(    ;
      O     DB327.DBX 1081.2;
      O     ;
      A     M   7503.4;
      AN    I      0.1;
      )     ;
      AN    M      3.3;
      =     M   7503.4;
      A     L      0.0;
      A(    ;
      O     DB327.DBX 1083.2;
      O     ;
      A     M   7503.5;
      AN    I      0.1;
      )     ;
      AN    M      3.3;
      =     M   7503.5;
NETWORK
TITLE =PROFINET ALARM-모듈이상이나 통신케이블단선(31~40)
//
//
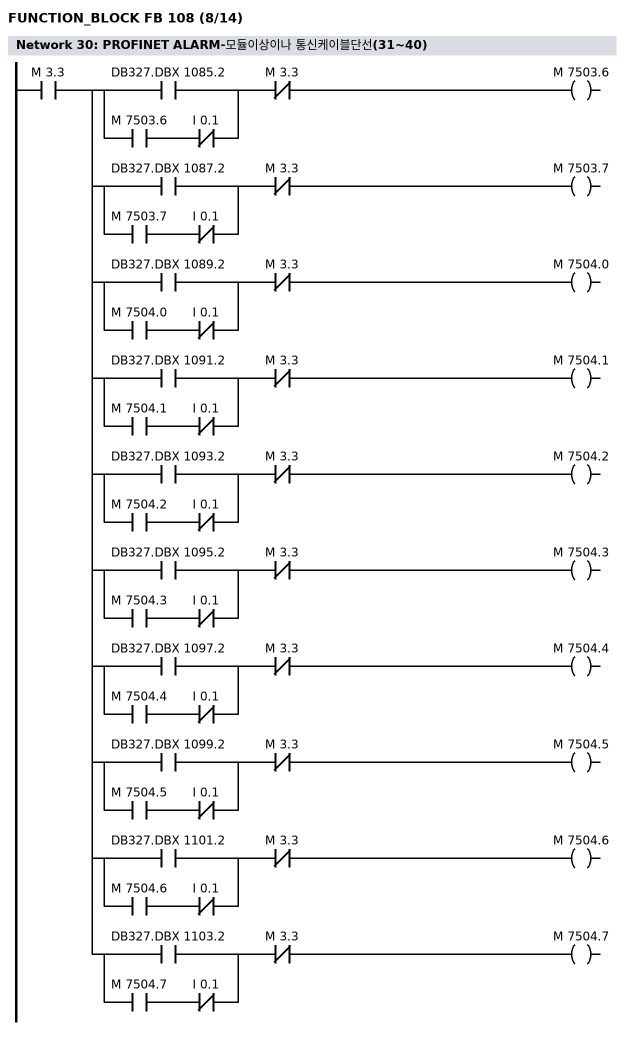
      A     M      3.3;
      =     L      0.0;
      A     L      0.0;
      A(    ;
      O     DB327.DBX 1085.2;
      O     ;
      A     M   7503.6;
      AN    I      0.1;
      )     ;
      AN    M      3.3;
      =     M   7503.6;
      A     L      0.0;
      A(    ;
      O     DB327.DBX 1087.2;
      O     ;
      A     M   7503.7;
      AN    I      0.1;
      )     ;
      AN    M      3.3;
      =     M   7503.7;
      A     L      0.0;
      A(    ;
      O     DB327.DBX 1089.2;
      O     ;
      A     M   7504.0;
      AN    I      0.1;
      )     ;
      AN    M      3.3;
      =     M   7504.0;
      A     L      0.0;
      A(    ;
      O     DB327.DBX 1091.2;
      O     ;
      A     M   7504.1;
      AN    I      0.1;
      )     ;
      AN    M      3.3;
      =     M   7504.1;
      A     L      0.0;
      A(    ;
      O     DB327.DBX 1093.2;
      O     ;
      A     M   7504.2;
      AN    I      0.1;
      )     ;
      AN    M      3.3;
      =     M   7504.2;
      A     L      0.0;
      A(    ;
      O     DB327.DBX 1095.2;
      O     ;
      A     M   7504.3;
      AN    I      0.1;
      )     ;
      AN    M      3.3;
      =     M   7504.3;
      A     L      0.0;
      A(    ;
      O     DB327.DBX 1097.2;
      O     ;
      A     M   7504.4;
      AN    I      0.1;
      )     ;
      AN    M      3.3;
      =     M   7504.4;
      A     L      0.0;
      A(    ;
      O     DB327.DBX 1099.2;
      O     ;
      A     M   7504.5;
      AN    I      0.1;
      )     ;
      AN    M      3.3;
      =     M   7504.5;
      A     L      0.0;
      A(    ;
      O     DB327.DBX 1101.2;
      O     ;
      A     M   7504.6;
      AN    I      0.1;
      )     ;
      AN    M      3.3;
      =     M   7504.6;
      A     L      0.0;
      A(    ;
      O     DB327.DBX 1103.2;
      O     ;
      A     M   7504.7;
      AN    I      0.1;
      )     ;
      AN    M      3.3;
      =     M   7504.7;
NETWORK
TITLE =PROFINET ALARM-모듈이상이나 통신케이블단선(150~159)
